(* CoDeSys 2.3.9.50 project: dacha.pro *)
(* Libraries: standard.lib 5.6.98 11:03:02, TcpIp.lib 9.1.14 13:33:22, TcBase.lib 14.5.09 11:14:08, TcSystem.lib 7.6.16 10:01:22, ModbusRTU.lib 13.5.15 12:38:16, TcIoFunctions.lib 27.1.17 16:22:22, COMlibV2.lb6 25.2.14 08:37:08, TcUtilities.lib 3.2.16 15:08:58 *)

(* Task configuration *)
TASK Standard (PRIORITY := 0, INTERVAL := T#50ms);
	MAIN
END_TASK

(* Global variable list: Global_Variables *)
VAR_GLOBAL


	Clear					: ClearComBuffer;
	MB						: ModbusRtuMaster_KL6x22B;
	TxBufferCom1			: ComBuffer;
	RxBufferCom1			: ComBuffer;
	SerialLineControlCom1		: SerialLineControl;
	ReceiveDataCom1		: ReceiveData;
	SendDataCom1			: SendData;
	Merc_address			: BYTE:=97;
	Sensor_CO2_high	 		: BYTE;	(*Старший байт датчика MH-Z19B*)
	Sensor_CO2_low 			: BYTE;	(*Младший байт датчика MH-Z19B*)
	iobroker					: iobroker_Struct;
	MB_vars					: stMB;
	Mercury					: stMercury;


	HW_temp_first_floor					AT %IW40:WORD;	(* Датчик температуры 1 этаж *)
	HW_temp_second_floor				AT %IW42:WORD;	(* Датчик температуры 2 этаж *)
	HW_temp_underfloor					AT %IW44:WORD;	(* Датчик температуры подпол 1 этаж *)
	HW_temp_sport						AT %IW46:WORD;	(* Датчик температуры спортзал *)

	HW_temp_sport_underfloor				AT %IW48:WORD;	(* Датчик температуры подпол спортзал *)
	HW_temp_sauna						AT %IW50:WORD;	(* Датчик температуры сауна*)
	HW_temp_street						AT %IW52:WORD;	(* Датчик температуры улица *)
	HW_temp_vent						AT %IW54:WORD;	(* Датчик температуры притока вентиляции *)

	HW_PIR_terrasa						AT %IX56.0:BOOL;		(*PIR датчик терраса *)
	HW_PIR_zapad						AT %IX56.1:BOOL;		(*PIR датчик запад *)
	HW_PIR_vostok						AT %IX56.2:BOOL;		(*PIR датчик восток *)
	HW_PIR_sport						AT %IX56.3:BOOL;		(*PIR датчик спортзал *)

	HW_GERKON_drovnik					AT %IX56.4:BOOL;		(*Геркон дровник *)
	HW_GERKON_door					AT %IX56.5:BOOL;		(*Геркон дверь *)
	HW_sensor_smoke_1floor				AT %IX56.6:BOOL;		(*Датчик дыма 1 этаж *)
	HW_sensor_smoke_2floor				AT %IX56.7:BOOL;		(*Датчик дыма 2 этаж *)

	HW_button_light_terrasa				AT %IX57.0:BOOL;		(* Кнопка прожектор терраса  *)
	HW_button_security					AT %IX57.1:BOOL;		(* Кнопка охрана  *)
	HW_button_vorota						AT %IX57.2:BOOL;		(* Кнопка открытия ворот  *)
	HW_button_kalitka					AT %IX57.3:BOOL;		(* Кнопка открытия калитки  *)

	HW_button_poliv_terrasa				AT %IX57.4:BOOL;		(* Кнопка полив терраса 2 часа  *)
	HW_button_poliv_zapad				AT %IX57.5:BOOL;		(* Кнопка полив запад  2 часа  *)
	HW_button_poliv_south				AT %IX57.6:BOOL;		(* Кнопка полив юг 2 часа  *)
(*	HW_reserved						AT %IX57.7:BOOL;	*)	(*   *)

	HW_sensor_supply					AT %IX58.0:BOOL;		(* Датчик напряжение  *)


	HW_heat_first_floor					AT %QX0.0:BOOL;		(* Отопление 1 этаж *)
	HW_heat_second_floor				AT %QX0.1:BOOL;		(* Отопление 2 этаж *)
	HW_heat_sport						AT %QX0.2:BOOL;		(* Отопление спортзал *)
	HW_heat_underfloor					AT %QX0.3:BOOL;		(* Отопление подпол *)
	HW_heat_sauna						AT %QX0.4:BOOL;		(* Отопление сауна *)
	HW_heat_bathroom					AT %QX0.5:BOOL;		(* Отопление душевая *)
	HW_heat_pipe						AT %QX0.6:BOOL;		(* Отопление водопровод *)
	HW_vent_underfloor					AT %QX0.7:BOOL;		(* Вентиляция подпола *)

	HW_vorota							AT %QX1.0:BOOL;		(* Ворота *)
	HW_kalitka							AT %QX1.1:BOOL;		(* Калитка *)
	HW_pomp_house						AT %QX1.2:BOOL;		(* Насос водоснабжения дома *)
	HW_pomp_garden					AT %QX1.3:BOOL;		(* Насос полива *)
	HW_light_garden						AT %QX1.4:BOOL;		(* Прожектор двор *)
	HW_light_terrasa						AT %QX1.5:BOOL;		(* Свет терраса *)
	HW_switch_security					AT %QX1.6:BOOL;		(* Реле охрана *)
	HW_switch_RS485					AT %QX1.7:BOOL:=TRUE;		(* RS485 line *)


	HW_vent_valve_input					AT %QX2.0:BOOL;		(* Клапан приточной вентиляции *)
	HW_vent_valve_output					AT %QX2.1:BOOL;		(* Клапан вытяжной вентиляции *)
	HW_trans_power						AT %QX2.2:BOOL;		(*Подача тока на трансформатор и реле ТЭН-а *)
	HW_vent_in_heat						AT %QX2.3:BOOL;		(* Подогрев притока - ТЭН *)
	HW_vent_in_heat_level				AT %QX2.4:BOOL;		(* Подогрев притока ночной режим   -5 К ТЭН *)
	HW_vent_in_trans_105_130				AT %QX2.5:BOOL:=FALSE;  (* Напряжение 110 или 130 В *)
	HW_vent_in_trans_160_220				AT %QX2.6:BOOL:=FALSE;  (* Напряжение 160 или 220 В *)
	HW_vent_in_trans_LO_HI				AT %QX2.7:BOOL:=FALSE;  (* Напряжение 110/130  или 160/220 В *)

	HW_poliv_terrasa						AT %QX3.0:BOOL;		(* полив терраса  *)
	HW_poliv_zapad						AT %QX3.1:BOOL;		(* полив запад   *)
	HW_poliv_south						AT %QX3.2:BOOL;		(* полив юг   *)


END_VAR

(* Global variable list: Global_Variables_persistent *)
VAR_GLOBAL PERSISTENT

	(*USER VARIABLES NEED TO BE ATTACHED TO %Q TO ENABLE SAVE IT IN NOVRAM, FOR CX ONLY *)

	Target_CO2_mem					AT %Q*:		INT;

	First_floor_temp_target_mem		AT %Q*:		INT;
	Second_floor_temp_target_mem		AT %Q*:		INT;
	Sport_temp_target_mem			AT %Q*:		INT;
	Sauna_temp_target_mem			AT %Q*:		INT;
	Underfloor_temp_target_mem		AT %Q*:		INT;
	Underfloor_humidity_target_mem	AT %Q*:		INT;

	Pomp_house_mem				AT %Q*:		BOOL;
	Pomp_garden_mem				AT %Q*:		BOOL;

	Light_garden_mem				AT %Q*:		BOOL;

	Vent_mem						AT %Q*:		BOOL;
	Vent_heat_mem					AT %Q*:		INT;
	Vent_heat_level_mem				AT %Q*:		BOOL;


END_VAR

(* Global variable list: TwinCAT_Configuration *)
(* Generated automatically by TwinCAT - (read only) *)
VAR_CONFIG
	.MB.InData AT %IB60 : MB_KL6inData22B;
	.MB.OutData AT %QB32 : MB_KL6outData22B;
	.Target_CO2_mem AT %QB6 : INT;
	.First_floor_temp_target_mem AT %QB56 : INT;
	.Second_floor_temp_target_mem AT %QB60 : INT;
	.Sport_temp_target_mem AT %QB62 : INT;
	.Sauna_temp_target_mem AT %QB72 : INT;
	.Underfloor_temp_target_mem AT %QB64 : INT;
	.Underfloor_humidity_target_mem AT %QB76 : INT;
	.Pomp_house_mem AT %QX68.0 : BOOL;
	.Pomp_garden_mem AT %QX74.0 : BOOL;
	.Light_garden_mem AT %QX66.1 : BOOL;
	.Vent_mem AT %QX28.0 : BOOL;
	.Vent_heat_mem AT %QB8 : INT;
	.Vent_heat_level_mem AT %QX28.3 : BOOL;
END_VAR

(* Global variable list: Variable_Configuration *)
VAR_CONFIG
	MB.InData AT %IB12 : MB_KL6inData22B;
	MB.OutData AT %QB12 : MB_KL6outData22B;

END_VAR

(* Data type *)
TYPE iobroker_Struct  :
STRUCT
	Vent_status				: 	INT;
	Valve_status				: 	INT;
	First_floor_temp 			:	REAL;
	First_floor_temp_target 		:	INT;
	First_floor_hum 			:	REAL;
	First_floor_CO2			:	REAL;
	Kitchen_room_temp		:	REAL;
	Kitchen_room_hum		:	REAL;
	Second_floor_temp 		:	REAL;
	Second_floor_temp_target 	:	INT;
	Second_floor_CO2 		:	REAL;
	Sport_temp	 			:	REAL;
	Sport_temp_target			:	INT;
	Sauna_temp	 			:	REAL;
	Sauna_temp_target		:	INT;
	Underfloor_temp			:	REAL;
	Underfloor_temp_target	:	INT;
	Underfloor_humidity		:	REAL;
	Underfloor_humidity_target	:	INT;
	Sport_underfloor_temp		:	REAL;
	Street_temp				:	REAL;
	Vent_temp				:	REAL;
	PIR_terrasa				:	BOOL:=TRUE;
	PIR_zapad				:	BOOL:=TRUE;
	PIR_vostok				:	BOOL:=TRUE;
	PIR_sport				:	BOOL:=TRUE;
	GERKON_drovnik			:	BOOL:=TRUE;
	Vent_input_level			:	INT;  (*  0-220 V  *)
	Vent_output_level			:	INT; (*0-100%*)
	Temp_vent_in			:	REAL;
	Vent_valve_status			:	INT;
	Security_status			:	BOOL;
	Target_CO2				:	INT;
	Vent						:	BOOL;
	Vent_underfloor			:	BOOL;
	Vent_out					:	BOOL;
	Vent_heat				:	INT;
	Vent_heat_level			:	BOOL;
	Vorota					:	BOOL;
	Vorota_open				:	BOOL;
	Kalitka					:	BOOL;
	Smoke					:	BOOL;
	Sensor_supply			:	BOOL;
	Pomp_house				:	BOOL;
	Pomp_garden			:	BOOL;
	Light_garden				:	BOOL;
	Poliv_zapad				:	BOOL;
	Poliv_terrasa				:	BOOL;
	Poliv_south				:	BOOL;
	Poliv_zapad_minutes		:	INT;
	Poliv_terrasa_minutes		:	INT;
	Poliv_south_minutes		:	INT;
	Uv1						:	REAL;
	Uv2						:	REAL;
	Uv3						:	REAL;
	Pw1						:	REAL;
	Pw2						:	REAL;
	Pw3						:	REAL;
	Pw_total					:	REAL;
	Ia1						:	REAL;
	Ia2						:	REAL;
	Ia3						:	REAL;
	E_T1					:	REAL;
	E_T2					:	REAL; (* 64 values*)

(*	M1T1					:	DWORD:=0;
	M1T2					:	DWORD:=0; (* 66 values*)

	M2T1					:	DWORD:=0; (* 67 values*)
	M2T2					:	DWORD:=0;
	M3T1					:	DWORD:=0;
	M3T2					:	DWORD:=0;
	M4T1					:	DWORD:=0; (* 70 values*)
	M4T2					:	DWORD:=0;
	M5T1					:	DWORD:=0;
	M5T2					:	DWORD:=0;
	M6T1					:	DWORD:=0;
	M6T2					:	DWORD:=0;
	M7T1					:	DWORD:=0;
	M7T2					:	DWORD:=0;
	M8T1					:	DWORD:=0;
	M8T2					:	DWORD:=0;
	M9T1					:	DWORD:=0;
	M9T2					:	DWORD:=0;
	M10T1					:	DWORD:=0;
	M10T2					:	DWORD:=0;
	M11T1					:	DWORD:=0;
	M11T2					:	DWORD:=0;
	M12T1					:	DWORD:=0;
	M12T2					:	DWORD:=0;   (* 86 values*)
*)

END_STRUCT
END_TYPE

(* Data type *)
(* @NESTEDCOMMENTS := 'Yes' *)
(* @PATH := '' *)
(* @OBJECTFLAGS := '0, 8' *)
TYPE ST_MqttReceivedPublishTelegram :
STRUCT
	sTopic		: STRING[255];
	sValue		: STRING[255];
	bHasData	: BOOL;
END_STRUCT
END_TYPE
(* @END_DECLARATION := '0' *)

(* Data type *)
(* @NESTEDCOMMENTS := 'Yes' *)
(* @PATH := '' *)
(* @OBJECTFLAGS := '0, 8' *)
TYPE ST_MqttSettings :
STRUCT
	(* informations *)
	sMqttClientId	: STRING[23];
	sMqttUserId	: STRING[25];
	sMqttPassword	: STRING[25];
	sMqttBrokerIP	: STRING[15];
	nMqttBrokerPort	: UDINT := 1883;

	(* state *)
	bSocketConnection	: BOOL := FALSE;
	bConnected			: BOOL := FALSE;
	bConnectPackageSent	: BOOL := FALSE;
	bDisconnect			: BOOL := FALSE;
	bError				: BOOL := FALSE;
	bValidConnection	: BOOL := FALSE;
	bActive				: BOOL := FALSE;
	wPackageIdentifier	: WORD := 1;
	hSocket				: T_HSOCKET;
	tonSendPingReq		: TON;

	(* send *)
	stMqttSendTelegram			: ST_MqttTelegram;
	stMqttLastSendTelegram		: ST_MqttTelegram;

	(* receive *)
	stMqttReceivedTelegram			: ST_MqttTelegram;
	stMqttLastReceivedTelegram		: ST_MqttTelegram;
	stMqttReceivedPublishTelegram	: ST_MqttReceivedPublishTelegram;

	(* settings internal *)
	iTelegramSize	: INT := 544;
	usKeepAliveTime	: USINT := 60; (* seconds *)

END_STRUCT
END_TYPE
(* @END_DECLARATION := '0' *)

(* Data type *)
(* @NESTEDCOMMENTS := 'Yes' *)
(* @PATH := '' *)
(* @OBJECTFLAGS := '0, 8' *)
TYPE ST_MqttTelegram :
STRUCT
	arMqttData 	: ARRAY[0..544] OF BYTE;
	nDataLength	: UDINT := 0;
END_STRUCT
END_TYPE
(* @END_DECLARATION := '0' *

(* Data type *)
TYPE stMB :
STRUCT

	M1T1							AT %MW0	:REAL;  (* modbus address 12288 *)
	M1T2							AT %MW4	:REAL;
	M2T1							AT %MW8	:REAL;
	M2T2							AT %MW12	:REAL;
	M3T1							AT %MW16	:REAL;
	M3T2							AT %MW20	:REAL;
	M4T1							AT %MW24	:REAL;
	M4T2							AT %MW28	:REAL;
	M5T1							AT %MW32	:REAL;
	M5T2							AT %MW36	:REAL;
	M6T1							AT %MW40	:REAL;
	M6T2							AT %MW44	:REAL;
	M7T1							AT %MW48	:REAL;
	M7T2							AT %MW52	:REAL;
	M8T1							AT %MW56	:REAL;
	M8T2							AT %MW60	:REAL;
	M9T1							AT %MW64	:REAL;
	M9T2							AT %MW68	:REAL;
	M10T1							AT %MW72	:REAL;
	M10T2							AT %MW76	:REAL;
	M11T1							AT %MW80	:REAL;
	M11T2							AT %MW84	:REAL;
	M12T1							AT %MW88	:REAL;
	M12T2							AT %MW92	:REAL;

END_STRUCT
END_TYPE

(* Data type *)
TYPE stMercury :
STRUCT

	M1T1					:	REAL;
	M1T2					:	REAL;
	M2T1					:	REAL;
	M2T2					:	REAL;
	M3T1					:	REAL;
	M3T2					:	REAL;
	M4T1					:	REAL;
	M4T2					:	REAL;
	M5T1					:	REAL;
	M5T2					:	REAL;
	M6T1					:	REAL;
	M6T2					:	REAL;
	M7T1					:	REAL;
	M7T2					:	REAL;
	M8T1					:	REAL;
	M8T2					:	REAL;
	M9T1					:	REAL;
	M9T2					:	REAL;
	M10T1					:	REAL;
	M10T2					:	REAL;
	M11T1					:	REAL;
	M11T2					:	REAL;
	M12T1					:	REAL;
	M12T2					:	REAL;

END_STRUCT
END_TYPE

(* POU MAIN, ST *)
PROGRAM MAIN
VAR

	INITVAR					: BOOL:=FALSE;

END_VAR
IF (INITVAR=FALSE) THEN

	(* START RESTORE VARS FROM MEMORY AFTER REBOOT/RESET/LOST POWER *)

	iobroker.Target_CO2				:=	Target_CO2_mem;
	iobroker.First_floor_temp_target		:=	First_floor_temp_target_mem;
	iobroker.Second_floor_temp_target	:=	Second_floor_temp_target_mem;
	iobroker.Sport_temp_target			:=	Sport_temp_target_mem;
	iobroker.Sauna_temp_target		:=	Sauna_temp_target_mem;

	iobroker.Underfloor_temp_target		:=	Underfloor_temp_target_mem;
	iobroker.Underfloor_humidity_target	:=	Underfloor_humidity_target_mem;
	iobroker.Vent						:=	Vent_mem;
	iobroker.Vent_heat				:=	Vent_heat_mem;
	iobroker.Vent_heat_level			:=	Vent_heat_level_mem;
	iobroker.Pomp_house				:=	Pomp_house_mem;
	iobroker.Pomp_garden				:=	Pomp_garden_mem;
	iobroker.Light_garden				:=	Light_garden_mem;
	(* END RESTORE VARS FROM MEMORY AFTER REBOOT/RESET/LOST POWER *)

	INITVAR:=TRUE;
ELSE
	(*START SAVE VARS to PERSISTENT MEMORY*)
	Target_CO2_mem					:=	iobroker.Target_CO2;
	First_floor_temp_target_mem		:=	iobroker.First_floor_temp_target;
	Second_floor_temp_target_mem		:=	iobroker.Second_floor_temp_target;
	Sport_temp_target_mem			:=	iobroker.Sport_temp_target;
	Underfloor_temp_target_mem		:=	iobroker.Underfloor_temp_target;
	Underfloor_humidity_target_mem	:=	iobroker.Underfloor_humidity_target;
	Vent_mem						:=	iobroker.Vent;
	Vent_heat_mem					:=	iobroker.Vent_heat;
	Vent_heat_level_mem				:=	iobroker.Vent_heat_level;
	Light_garden_mem				:=	iobroker.Light_garden;
	Pomp_house_mem				:=	iobroker.Pomp_house;
	(*END SAVE VARS to PERSISTENT MEMORY*)


	Sensors;						(* Аналогвые датчики на шине KL *)
	Security;						(* Мониторинг датчиков охраны *)
	RS485read;					(* Опрос устройств на шине RS485 *)
	Mqtt;						(* MQTT *)
	Thermocontrol;				(* Термостат*)
	VentControl;					(* Глобальный контроль вентустановки*)
	VentPower;					(* Авторегулировка мощности вентустановки по датчикам CO2*)
	Poliv;						(* Таймеры зонального полива *)


	(* Прямое присовение виртуальных переменных к переменным, жестко привязаным к физ. портам. Частота обновления= циклу ПЛК (50 мсек) : *)
	HW_vorota					:=	iobroker.Vorota;
	HW_kalitka					:=	iobroker.Kalitka;
	HW_pomp_house				:=	iobroker.Pomp_house;
	HW_light_garden				:=	iobroker.Light_garden;
	iobroker.Sensor_supply		:=	HW_sensor_supply;
	HW_vent_underfloor			:=	iobroker.Vent_underfloor;

END_IF
END_PROGRAM

(* POU Sensors, ST *)
PROGRAM Sensors
VAR
	Period_sensors_read		: INT:=30; (* Частота присвоения значений аналоговых температурных датчиков с модулей KL, секунды *)
	Timer					: TON;
	TimerQ					: BOOL;
	tTimerValue				: TIME;
END_VAR
Timer();

tTimerValue := DINT_TO_TIME(Period_sensors_read*1000);

	Timer(IN:=NOT TimerQ , PT:=tTimerValue , Q=>TimerQ , ET=> );
	IF timer.q THEN

		(*Temperature First_floor start*)
		iobroker.First_floor_temp:=WORD_TO_REAL(HW_temp_first_floor);
		IF (iobroker.First_floor_temp/10>1000)  THEN
			iobroker.First_floor_temp:=iobroker.First_floor_temp-65535;
			iobroker.First_floor_temp:=iobroker.First_floor_temp/10;
		ELSE
			iobroker.First_floor_temp:=iobroker.First_floor_temp/10;
		END_IF
		(*Temperature First_floor end*)

		(*Temperature second_floor start*)
		iobroker.Second_floor_temp:=WORD_TO_REAL(HW_temp_second_floor);
		IF (iobroker.Second_floor_temp/10>1000)  THEN
			iobroker.Second_floor_temp:=iobroker.Second_floor_temp-65535;
			iobroker.Second_floor_temp:=iobroker.Second_floor_temp/10;
		ELSE
			iobroker.Second_floor_temp:=iobroker.Second_floor_temp/10;
		END_IF
		(*Temperature second_floor end*)

		(*Temperature second_floor start*)
		iobroker.Sport_temp:=WORD_TO_REAL(HW_temp_sport);
		IF (iobroker.Sport_temp/10>1000)  THEN
			iobroker.Sport_temp:=iobroker.Sport_temp-65535;
			iobroker.Sport_temp:=iobroker.Sport_temp/10;
		ELSE
			iobroker.Sport_temp:=iobroker.Sport_temp/10;
		END_IF
		(*Temperature second_floor end*)

		(*Temperature street start*)
		iobroker.Street_temp:=WORD_TO_REAL(HW_temp_street);
		IF (iobroker.Street_temp/10>1000)  THEN
			iobroker.Street_temp:=iobroker.Street_temp-65535;
			iobroker.Street_temp:=iobroker.Street_temp/10;
		ELSE
			iobroker.Street_temp:=iobroker.Street_temp/10;
		END_IF
		(*Temperature street end*)

		(*Temperature vent start*)
		iobroker.Vent_temp:=WORD_TO_REAL(HW_temp_vent);
		IF (iobroker.Vent_temp/10>1000)  THEN
			iobroker.Vent_temp:=iobroker.Vent_temp-65535;
			iobroker.Vent_temp:=iobroker.Vent_temp/10;
		ELSE
			iobroker.Vent_temp:=iobroker.Vent_temp/10;
		END_IF
		(*Temperature vent end*)
	END_IF
END_PROGRAM

(* POU Security, ST *)
PROGRAM Security
VAR
	TRIG_PIR_terrasa			:	F_TRIG;
	TRIG_PIR_zapad			:	F_TRIG;
	TRIG_PIR_vostok			:	F_TRIG;
	TRIG_PIR_sport			:	F_TRIG;
	TRIG_GERKON_drovnik	:	F_TRIG;
	TRIG_sensor_smoke_1floor:	F_TRIG;

	trig_mem_terrasa				:	BOOL:=FALSE;
	trig_mem_zapad				:	BOOL:=FALSE;
	trig_mem_vostok				:	BOOL:=FALSE;
	trig_mem_sport				:	BOOL:=FALSE;
	trig_mem_drovnik				:	BOOL:=FALSE;
	trig_mem_sensor_smoke_1floor	:	BOOL:=FALSE;

END_VAR
(*  Используем триггеры для исключения ложной информации о сработке датчиков при перезагрузке ПЛК *)


TRIG_PIR_terrasa(CLK :=HW_PIR_terrasa);
TRIG_PIR_zapad(CLK :=HW_PIR_zapad);
TRIG_PIR_vostok(CLK :=HW_PIR_vostok);
TRIG_PIR_sport(CLK :=HW_PIR_sport);
TRIG_GERKON_drovnik(CLK :=HW_GERKON_drovnik);
TRIG_sensor_smoke_1floor(CLK :=HW_sensor_smoke_1floor);


IF (NOT TRIG_PIR_terrasa.Q) THEN
	iobroker.PIR_terrasa:=NOT TRIG_PIR_terrasa.Q;
END_IF
IF (trig_mem_terrasa=TRUE) THEN
	iobroker.PIR_terrasa:=FALSE;
	trig_mem_terrasa:=FALSE;
END_IF
IF (TRIG_PIR_terrasa.Q) THEN
	trig_mem_terrasa:=TRUE;
END_IF



IF (NOT TRIG_PIR_zapad.Q) THEN
	iobroker.PIR_zapad:=NOT TRIG_PIR_zapad.Q;
END_IF
IF (trig_mem_zapad=TRUE) THEN
	iobroker.PIR_zapad:=FALSE;
	trig_mem_zapad:=FALSE;
END_IF
IF (TRIG_PIR_zapad.Q) THEN
	trig_mem_zapad:=TRUE;
END_IF


IF (NOT TRIG_PIR_vostok.Q) THEN
	iobroker.PIR_vostok:=NOT TRIG_PIR_vostok.Q;
END_IF
IF (trig_mem_vostok=TRUE) THEN
	iobroker.PIR_vostok:=FALSE;
	trig_mem_vostok:=FALSE;
END_IF
IF (TRIG_PIR_vostok.Q) THEN
	trig_mem_vostok:=TRUE;
END_IF


IF (NOT TRIG_PIR_sport.Q) THEN
	iobroker.PIR_sport:=NOT TRIG_PIR_sport.Q;
END_IF
IF (trig_mem_sport=TRUE) THEN
	iobroker.PIR_sport:=FALSE;
	trig_mem_sport:=FALSE;
END_IF
IF (TRIG_PIR_sport.Q) THEN
	trig_mem_sport:=TRUE;
END_IF

IF (NOT TRIG_GERKON_drovnik.Q) THEN
	iobroker.GERKON_drovnik:=NOT TRIG_GERKON_drovnik.Q;
END_IF
IF (trig_mem_drovnik=TRUE) THEN
	iobroker.GERKON_drovnik:=FALSE;
	trig_mem_drovnik:=FALSE;
END_IF
IF (TRIG_GERKON_drovnik.Q) THEN
	trig_mem_drovnik:=TRUE;
END_IF


IF (NOT TRIG_sensor_smoke_1floor.Q) THEN
	iobroker.SMOKE:=NOT TRIG_sensor_smoke_1floor.Q;
END_IF
IF (trig_mem_sensor_smoke_1floor=TRUE) THEN
	iobroker.SMOKE:=FALSE;
	trig_mem_sensor_smoke_1floor:=FALSE;
END_IF
IF (TRIG_sensor_smoke_1floor.Q) THEN
	trig_mem_sensor_smoke_1floor:=TRUE;
END_IF
END_PROGRAM

(* POU RS485read, ST *)
PROGRAM RS485read
VAR

	password_1				: ARRAY [1..6] OF BYTE:=6(1); (* пароль к меркуриям, по умолчанию 6 единиц*)
	crctest					: WORD;
	arrReceive				: ARRAY[1..22] OF BYTE;
	arrSend					: ARRAY[1..22] OF BYTE;

	MBdata_kitchen			 : ARRAY [1..2] OF WORD;
	FtrigBusy				: F_TRIG;
	timeoutvalue				: TIME := T#500ms;		(* timeout while waiting for an answer of the modbus slave *)
	state					: INT;
	busy					: BOOL;
	LastErrorstate				: INT;
	LastModbusError			: ST_ModbusErrorDiagnostics;
	CounterError				: DINT;
	CounterSuccess			: DINT;
	Timer1					: TON;
	Timer1Q					: BOOL;
	Timer_day				:TON;
	Timer_dayQ				:BOOL;

	tmCheck					:TON;

	get_co2_mh_z19b_1floor	: FB_GET_CO2_MH_Z19B;
	get_co2_mh_z19b_2floor	: FB_GET_CO2_MH_Z19B;
	get_supply				: FB_GET_SUPPLY;
	get_current				: FB_GET_CURRENT;
	get_power				: FB_GET_POWER;
	get_energy_E_T1			: FB_GET_ENERGY;
	get_energy_E_T2			: FB_GET_ENERGY;
	get_energy_M1T1			: FB_GET_ENERGY;
	get_energy_M1T2			: FB_GET_ENERGY;
	get_energy_M2T1			: FB_GET_ENERGY;
	get_energy_M2T2			: FB_GET_ENERGY;
	get_energy_M3T1			: FB_GET_ENERGY;
	get_energy_M3T2			: FB_GET_ENERGY;
	get_energy_M4T1			: FB_GET_ENERGY;
	get_energy_M4T2			: FB_GET_ENERGY;
	get_energy_M5T1			: FB_GET_ENERGY;
	get_energy_M5T2			: FB_GET_ENERGY;
	get_energy_M6T1			: FB_GET_ENERGY;
	get_energy_M6T2			: FB_GET_ENERGY;
	get_energy_M7T1			: FB_GET_ENERGY;
	get_energy_M7T2			: FB_GET_ENERGY;
	get_energy_M8T1			: FB_GET_ENERGY;
	get_energy_M8T2			: FB_GET_ENERGY;
	get_energy_M9T1			: FB_GET_ENERGY;
	get_energy_M9T2			: FB_GET_ENERGY;
	get_energy_M10T1		: FB_GET_ENERGY;
	get_energy_M10T2		: FB_GET_ENERGY;
	get_energy_M11T1		: FB_GET_ENERGY;
	get_energy_M11T2		: FB_GET_ENERGY;
	get_energy_M12T1		: FB_GET_ENERGY;
	get_energy_M12T2		: FB_GET_ENERGY;

	get_co2_mh_z19b_1floor_done	: BOOL;
	get_co2_mh_z19b_2floor_done	: BOOL;
	get_supply_done			: BOOL;
	get_current_done			: BOOL;
	get_power_done			: BOOL;
	get_energy_E_T1_done	: BOOL;
	get_energy_E_T2_done	: BOOL;
	get_energy_M1T1_done	: BOOL;
	get_energy_M1T2_done	: BOOL;
	get_energy_M2T1_done	: BOOL;
	get_energy_M2T2_done	: BOOL;
	get_energy_M3T1_done	: BOOL;
	get_energy_M3T2_done	: BOOL;
	get_energy_M4T1_done	: BOOL;
	get_energy_M4T2_done	: BOOL;
	get_energy_M5T1_done	: BOOL;
	get_energy_M5T2_done	: BOOL;
	get_energy_M6T1_done	: BOOL;
	get_energy_M6T2_done	: BOOL;
	get_energy_M7T1_done	: BOOL;
	get_energy_M7T2_done	: BOOL;
	get_energy_M8T1_done	: BOOL;
	get_energy_M8T2_done	: BOOL;
	get_energy_M9T1_done	: BOOL;
	get_energy_M9T2_done	: BOOL;
	get_energy_M10T1_done	: BOOL;
	get_energy_M10T2_done	: BOOL;
	get_energy_M11T1_done	: BOOL;
	get_energy_M11T2_done	: BOOL;
	get_energy_M12T1_done	: BOOL;
	get_energy_M12T2_done	: BOOL;
END_VAR

VAR_INPUT


END_VAR
tmCheck();
Timer_day();

CASE state OF
	0:
		MB.ReadRegs(Execute:= FALSE);

		state := 1;
	1:	(* Read Temp and Hum data  from sensor *)
		Clear(Buffer := RxBufferCom1);
		MB.ReadRegs(
			UnitID:= 16#07, (* station address *)
			Quantity:= 2,	(* WORDs *)
			MBAddr:= 0,
			cbLength:= 6,
			pMemoryAddr:= ADR(MBdata_kitchen),
			Execute:= TRUE,
			Timeout:= timeoutvalue,
			Busy => busy,
		);
		IF NOT busy THEN
			IF (mb.Error = FALSE ) THEN
				iobroker.Kitchen_room_temp:=WORD_TO_REAL(MBdata_kitchen[1])/10;
				iobroker.Kitchen_room_hum:=WORD_TO_REAL(MBdata_kitchen[2])/10;
				MB.ReadRegs(Execute:= FALSE);
				state := 2;
			END_IF
			MB.ReadRegs(Execute:= FALSE);
			state :=2;
		END_IF

2:	(* Read CO2 from sensor *)

		tmCheck(in:=FALSE);
		tmCheck(in:=TRUE,pt:=t#2s);
		get_co2_mh_z19b_1floor_done := FALSE;
		get_co2_mh_z19b_1floor( co2=>iobroker.First_Floor_CO2, done=>get_co2_mh_z19b_1floor_done);
		IF get_co2_mh_z19b_1floor_done = TRUE THEN
			state:=3;
		ELSIF tmcheck.Q THEN
			 state:=3;
		END_IF

3:
	HW_switch_RS485:=TRUE;
	Timer1(IN:=NOT Timer1Q , PT:=T#1s , Q=>Timer1Q , ET=> );
	IF timer1.q THEN
		state:=4;
	END_IF

4:

		tmCheck(in:=FALSE);
		tmCheck(in:=TRUE,pt:=t#2s);
		get_co2_mh_z19b_2floor_done := FALSE;
		get_co2_mh_z19b_2floor( co2=>iobroker.Second_Floor_CO2, done=>get_co2_mh_z19b_2floor_done);
		IF get_co2_mh_z19b_2floor_done = TRUE THEN
			state:=41;
		ELSIF tmcheck.Q THEN
			 state:=41;
		END_IF



41:
	Timer1(IN:=NOT Timer1Q , PT:=T#2s , Q=>Timer1Q , ET=> );
	IF timer1.q THEN
	HW_switch_RS485:=FALSE;
		state:=5;
	END_IF

5: (*открываем канал*)


	Clear(Buffer := RxBufferCom1);
	arrSend[1]:=Merc_address;
	arrSend[2]:=1; (*код доступа*)
	arrSend[3]:=1; (*Уровень доступа*)

	MEMCPY(ADR(arrSend)+3,ADR(password_1),6); (*пароль*)
	crctest:=F_CRC16(ADR(arrSend),9); (*расчет контрольной суммы*)
	MEMCPY(ADR(arrSend)+9,ADR(crctest),SIZEOF(crctest)); (*прибавление контрольной суммы к запросу*)
	SendDataCom1(pSendData:=ADR(arrSend),Length:=11,TXBuffer:=TxBufferCom1,Busy=>,Error=>);
	tmCheck(in:=FALSE); tmCheck(in:=TRUE,pt:=t#2s); 	(*запуск таймера проверки - потеря связи\обрыв кабеля*)
	state:=6;

6: (*ответ*)
	ReceiveDataCom1(pPrefix:=,LenPrefix:=,pSuffix:=,LenSuffix:=,
	pReceiveData:=ADR(arrReceive),SizeReceiveData:=4,
	Timeout:=t#2s,Reset:=,
	RXbuffer:=RxBufferCom1,
	DataReceived=>,busy=>,Error=>,RxTimeout=>,LenReceiveData=>);
	IF ReceiveDataCom1.Error <> 0 THEN state:=888; END_IF
	IF receiveDataCom1.DataReceived THEN state:=7;
	ELSIF tmcheck.Q THEN state:=888;
	END_IF
7: (*проверка ответа*)

	IF arrReceive[1] = Merc_address THEN state:= 8;
	ELSE	state:=888;
	END_IF



8:
		tmCheck(in:=FALSE);
		tmCheck(in:=TRUE,pt:=t#2s);
		get_supply_done := FALSE;
		get_supply( byte1:=16#8, byte2:=16#16, byte3:=16#11,  supply1=>iobroker.UV1,supply2=>iobroker.UV2,supply3=>iobroker.UV3, done=>get_supply_done);
		IF get_supply_done = TRUE THEN
			state:=9;
		ELSIF tmcheck.Q THEN
			 state:=888;
		END_IF

 (*запрос на чтение тока  на всех фазах
--------------------------------------------------------------------------------------------------------------------------------------------------------------------
*)
9:
		tmCheck(in:=FALSE);
		tmCheck(in:=TRUE,pt:=t#2s);
		get_current_done := FALSE;
		get_current(byte1:=16#8, byte2:=16#16, byte3:=16#21,  current1=>iobroker.Ia1,current2=>iobroker.Ia2,current3=>iobroker.Ia3, done=>get_current_done);
		IF get_current_done = TRUE THEN
			state:=10;
		ELSIF tmcheck.Q THEN state:=888;
		END_IF

 (*запрос на чтение мощности  на всех фазах
--------------------------------------------------------------------------------------------------------------------------------------------------------------------
*)

10:
		tmCheck(in:=FALSE);
		tmCheck(in:=TRUE,pt:=t#2s);
		get_power_done := FALSE;
		get_power(byte1:=16#8, byte2:=16#16, byte3:=16#0,  power_total=>iobroker.pw_total, power1=>iobroker.pw1, power2=>iobroker.pw2,power3=>iobroker.pw3,done=>get_power_done);
		IF get_power_done = TRUE THEN
			state:=11;
		ELSIF tmcheck.Q THEN state:=888;
		END_IF

 (*запрос на чтение энергии T1
--------------------------------------------------------------------------------------------------------------------------------------------------------------------
*)
11:
	tmCheck(in:=FALSE);
		tmCheck(in:=TRUE,pt:=t#2s);
		get_energy_E_T1_done := FALSE;
		get_energy_E_T1(byte1:=5, byte2:=16#0, byte3:=1,  energy=>iobroker.E_T1, done=>get_energy_E_T1_done);
		IF get_energy_E_T1_done = TRUE THEN
			state:=12;
		ELSIF tmcheck.Q THEN state:=888;
		END_IF
 (*запрос на чтение энергии T2
--------------------------------------------------------------------------------------------------------------------------------------------------------------------
*)

12:
	tmCheck(in:=FALSE);
		tmCheck(in:=TRUE,pt:=t#2s);
		get_energy_E_T2_done := FALSE;
		get_energy_E_T2(byte1:=5, byte2:=16#0, byte3:=2,  energy=>iobroker.E_T2, done=>get_energy_E_T2_done);
		IF get_energy_E_T2_done = TRUE THEN
			state:=13;
		ELSIF tmcheck.Q THEN state:=888;
		END_IF


13:
		Timer_day(IN:=NOT Timer_dayQ , PT:=T#10m , Q=>Timer_dayQ , ET=> );
			IF timer_day.q THEN
				state:=14;
			ELSE
				state:=888;
			END_IF

14:
		tmCheck(in:=FALSE);
		tmCheck(in:=TRUE,pt:=t#2s);
		get_energy_M1T1_done := FALSE;
		get_energy_M1T1(byte1:=5, byte2:=16#31, byte3:=1,   energy=>MB_vars.M1T1,done=>get_energy_M1T1_done);
		IF get_energy_M1T1_done = TRUE THEN
			Mercury.M1T1:=MB_vars.M1T1;
			state:=15;
		ELSIF tmcheck.Q THEN state:=888;
		END_IF
15:
		tmCheck(in:=FALSE);
		tmCheck(in:=TRUE,pt:=t#2s);
		get_energy_M1T2_done := FALSE;
		get_energy_M1T2(byte1:=5, byte2:=16#31, byte3:=2,energy=>MB_vars.M1T2,done=>get_energy_M1T2_done);
		IF get_energy_M1T2_done = TRUE THEN
			Mercury.M1T2:=MB_vars.M1T2;
			state:=16;
		ELSIF tmcheck.Q THEN state:=888;
		END_IF

16:
		tmCheck(in:=FALSE);
		tmCheck(in:=TRUE,pt:=t#2s);
		get_energy_M2T1_done := FALSE;
		get_energy_M2T1(byte1:=5, byte2:=16#32, byte3:=1, energy=>MB_vars.M2T1, done=>get_energy_M2T1_done);
		IF get_energy_M2T1_done = TRUE THEN
			Mercury.M2T1:=MB_vars.M2T1;
			state:=17;
		ELSIF tmcheck.Q THEN state:=888;
		END_IF
17:
		tmCheck(in:=FALSE);
		tmCheck(in:=TRUE,pt:=t#2s);
		get_energy_M2T2_done := FALSE;
		get_energy_M2T2(byte1:=5, byte2:=16#32, byte3:=2, energy=>MB_vars.M2T2,done=>get_energy_M2T2_done);
		IF get_energy_M2T2_done = TRUE THEN
			Mercury.M2T2:=MB_vars.M2T2;
			state:=18;
		ELSIF tmcheck.Q THEN state:=888;
		END_IF
18:
		tmCheck(in:=FALSE);
		tmCheck(in:=TRUE,pt:=t#2s);
		get_energy_M3T1_done := FALSE;
		get_energy_M3T1(byte1:=5, byte2:=16#33, byte3:=1, energy=>MB_vars.M3T1, done=>get_energy_M3T1_done);
		IF get_energy_M3T1_done = TRUE THEN
			Mercury.M3T1:=MB_vars.M3T1;
			state:=19;
		ELSIF tmcheck.Q THEN state:=888;
		END_IF
19:
		tmCheck(in:=FALSE);
		tmCheck(in:=TRUE,pt:=t#2s);
		get_energy_M3T2_done := FALSE;
		get_energy_M3T2(byte1:=5, byte2:=16#33, byte3:=2, energy=>MB_vars.M3T2,done=>get_energy_M3T2_done);
		IF get_energy_M3T2_done = TRUE THEN
			Mercury.M3T2:=MB_vars.M3T2;
			state:=20;
		ELSIF tmcheck.Q THEN state:=888;
		END_IF
20:
		tmCheck(in:=FALSE);
		tmCheck(in:=TRUE,pt:=t#2s);
		get_energy_M4T1_done := FALSE;
		get_energy_M4T1(byte1:=5, byte2:=16#34, byte3:=1, energy=>MB_vars.M4T1, done=>get_energy_M4T1_done);
		IF get_energy_M4T1_done = TRUE THEN
			Mercury.M4T1:=MB_vars.M4T1;
			state:=21;
		ELSIF tmcheck.Q THEN state:=888;
		END_IF
21:
		tmCheck(in:=FALSE);
		tmCheck(in:=TRUE,pt:=t#2s);
		get_energy_M4T2_done := FALSE;
		get_energy_M4T2(byte1:=5, byte2:=16#34, byte3:=2, energy=>MB_vars.M4T2,done=>get_energy_M4T2_done);
		IF get_energy_M4T2_done = TRUE THEN
			Mercury.M4T2:=MB_vars.M4T2;
			state:=22;
		ELSIF tmcheck.Q THEN state:=888;
		END_IF
22:
		tmCheck(in:=FALSE);
		tmCheck(in:=TRUE,pt:=t#2s);
		get_energy_M5T1_done := FALSE;
		get_energy_M5T1(byte1:=5, byte2:=16#35, byte3:=1, energy=>MB_vars.M5T1, done=>get_energy_M5T1_done);
		IF get_energy_M5T1_done = TRUE THEN
			Mercury.M5T1:=MB_vars.M5T1;
			state:=23;
		ELSIF tmcheck.Q THEN state:=888;
		END_IF
23:
		tmCheck(in:=FALSE);
		tmCheck(in:=TRUE,pt:=t#2s);
		get_energy_M5T2_done := FALSE;
		get_energy_M5T2(byte1:=5, byte2:=16#35, byte3:=2, energy=>MB_vars.M5T2,done=>get_energy_M5T2_done);
		IF get_energy_M5T2_done = TRUE THEN
			Mercury.M5T2:=MB_vars.M5T2;
			state:=24;
		ELSIF tmcheck.Q THEN state:=888;
		END_IF
24:
		tmCheck(in:=FALSE);
		tmCheck(in:=TRUE,pt:=t#2s);
		get_energy_M6T1_done := FALSE;
		get_energy_M6T1(byte1:=5, byte2:=16#36, byte3:=1, energy=>MB_vars.M6T1, done=>get_energy_M6T1_done);
		IF get_energy_M6T1_done = TRUE THEN
			Mercury.M6T1:=MB_vars.M6T1;
			state:=25;
		ELSIF tmcheck.Q THEN state:=888;
		END_IF
25:
		tmCheck(in:=FALSE);
		tmCheck(in:=TRUE,pt:=t#2s);
		get_energy_M6T2_done := FALSE;
		get_energy_M6T2(byte1:=5, byte2:=16#36, byte3:=2, energy=>MB_vars.M6T2,done=>get_energy_M6T2_done);
		IF get_energy_M6T2_done = TRUE THEN
			Mercury.M6T2:=MB_vars.M6T2;
			state:=26;
		ELSIF tmcheck.Q THEN state:=888;
		END_IF
26:
		tmCheck(in:=FALSE);
		tmCheck(in:=TRUE,pt:=t#2s);
		get_energy_M7T1_done := FALSE;
		get_energy_M7T1(byte1:=5, byte2:=16#37, byte3:=1, energy=>MB_vars.M7T1, done=>get_energy_M7T1_done);
		IF get_energy_M7T1_done = TRUE THEN
			Mercury.M7T1:=MB_vars.M7T1;
			state:=27;
		ELSIF tmcheck.Q THEN state:=888;
		END_IF
27:
		tmCheck(in:=FALSE);
		tmCheck(in:=TRUE,pt:=t#2s);
		get_energy_M7T2_done := FALSE;
		get_energy_M7T2(byte1:=5, byte2:=16#37, byte3:=2, energy=>MB_vars.M7T2,done=>get_energy_M7T2_done);
		IF get_energy_M7T2_done = TRUE THEN
			Mercury.M7T2:=MB_vars.M7T2;
			state:=28;
		ELSIF tmcheck.Q THEN state:=888;
		END_IF
28:
		tmCheck(in:=FALSE);
		tmCheck(in:=TRUE,pt:=t#2s);
		get_energy_M8T1_done := FALSE;
		get_energy_M8T1(byte1:=5, byte2:=16#38, byte3:=1, energy=>MB_vars.M8T1, done=>get_energy_M8T1_done);
		IF get_energy_M8T1_done = TRUE THEN
			Mercury.M8T1:=MB_vars.M8T1;
			state:=29;
		ELSIF tmcheck.Q THEN state:=888;
		END_IF
29:
		tmCheck(in:=FALSE);
		tmCheck(in:=TRUE,pt:=t#2s);
		get_energy_M8T2_done := FALSE;
		get_energy_M8T2(byte1:=5, byte2:=16#38, byte3:=2, energy=>MB_vars.M8T2,done=>get_energy_M8T2_done);
		IF get_energy_M8T2_done = TRUE THEN
			Mercury.M8T2:=MB_vars.M8T2;
			state:=30;
		ELSIF tmcheck.Q THEN state:=888;
		END_IF
30:
		tmCheck(in:=FALSE);
		tmCheck(in:=TRUE,pt:=t#2s);
		get_energy_M9T1_done := FALSE;
		get_energy_M9T1(byte1:=5, byte2:=16#39, byte3:=1, energy=>MB_vars.M9T1, done=>get_energy_M9T1_done);
		IF get_energy_M9T1_done = TRUE THEN
			Mercury.M9T1:=MB_vars.M9T1;
			state:=31;
		ELSIF tmcheck.Q THEN state:=888;
		END_IF
31:
		tmCheck(in:=FALSE);
		tmCheck(in:=TRUE,pt:=t#2s);
		get_energy_M9T2_done := FALSE;
		get_energy_M9T2(byte1:=5, byte2:=16#39, byte3:=2,  energy=>MB_vars.M9T2,done=>get_energy_M9T2_done);
		IF get_energy_M9T2_done = TRUE THEN
			Mercury.M9T2:=MB_vars.M9T2;
			state:=32;
		ELSIF tmcheck.Q THEN state:=888;
		END_IF
32:
		tmCheck(in:=FALSE);
		tmCheck(in:=TRUE,pt:=t#2s);
		get_energy_M10T1_done := FALSE;
		get_energy_M10T1(byte1:=5, byte2:=16#3A, byte3:=1,  energy=>MB_vars.M10T1, done=>get_energy_M10T1_done);
		IF get_energy_M10T1_done = TRUE THEN
			Mercury.M10T1:=MB_vars.M10T1;
			state:=33;
		ELSIF tmcheck.Q THEN state:=888;
		END_IF
33:
		tmCheck(in:=FALSE);
		tmCheck(in:=TRUE,pt:=t#2s);
		get_energy_M10T2_done := FALSE;
		get_energy_M10T2(byte1:=5, byte2:=16#3A, byte3:=2, energy=>MB_vars.M10T2,done=>get_energy_M10T2_done);
		IF get_energy_M10T2_done = TRUE THEN
			Mercury.M10T2:=MB_vars.M10T2;
			state:=34;
		ELSIF tmcheck.Q THEN state:=888;
		END_IF
34:
		tmCheck(in:=FALSE);
		tmCheck(in:=TRUE,pt:=t#2s);
		get_energy_M11T1_done := FALSE;
		get_energy_M11T1(byte1:=5, byte2:=16#3B, byte3:=1,  energy=>MB_vars.M11T1, done=>get_energy_M11T1_done);
		IF get_energy_M11T1_done = TRUE THEN
			Mercury.M11T1:=MB_vars.M11T1;
			state:=35;
		ELSIF tmcheck.Q THEN state:=888;
		END_IF
35:
		tmCheck(in:=FALSE);
		tmCheck(in:=TRUE,pt:=t#2s);
		get_energy_M11T2_done := FALSE;
		get_energy_M11T2(byte1:=5, byte2:=16#3B, byte3:=2, energy=>MB_vars.M11T2,done=>get_energy_M11T2_done);
		IF get_energy_M11T2_done = TRUE THEN
			Mercury.M11T2:=MB_vars.M11T2;
			state:=36;
		ELSIF tmcheck.Q THEN state:=888;
		END_IF
36:
		tmCheck(in:=FALSE);
		tmCheck(in:=TRUE,pt:=t#2s);
		get_energy_M12T1_done := FALSE;
		get_energy_M12T1(byte1:=5, byte2:=16#3C, byte3:=1,  energy=>MB_vars.M12T1, done=>get_energy_M12T1_done);
		IF get_energy_M12T1_done = TRUE THEN
			Mercury.M12T1:=MB_vars.M12T1;
			state:=37;
		ELSIF tmcheck.Q THEN state:=888;
		END_IF
37:
		tmCheck(in:=FALSE);
		tmCheck(in:=TRUE,pt:=t#2s);
		get_energy_M12T2_done := FALSE;
		get_energy_M12T2(byte1:=5, byte2:=16#3C, byte3:=2,  energy=>MB_vars.M12T2,done=>get_energy_M12T2_done);
		IF get_energy_M12T2_done = TRUE THEN
			Mercury.M12T2:=MB_vars.M12T2;
			state:=888;
		ELSIF tmcheck.Q THEN state:=888;
		END_IF



888:
		Timer1(IN:=NOT Timer1Q , PT:=T#60s , Q=>Timer1Q , ET=> );
		IF timer1.q THEN

		state:=0;
		END_IF

END_CASE

FtrigBusy(CLK:=mb.BUSY );
IF FtrigBusy.Q THEN
	IF mb.Error THEN
		LastModbusError := mb.ErrorDiagnostics;
		LastErrorstate := state;
		CounterError := CounterError + 1;
	ELSE
		CounterSuccess := CounterSuccess + 1;
	END_IF
END_IF



SerialLinecontrolCom1(
	mode:=SerialLinemode_kl6_22b_standard,
	pComIn:=ADR(RS485read.MB.InData),
	pComOut:=ADR(RS485read.MB.OutData),
	SizeComIn:=SIZEOF(RS485read.MB.OutData),
	TxBuffer:=TxBufferCom1,
	RxBuffer:=RxBufferCom1,
	Error=>,
	errorid=>);
END_PROGRAM

(* POU FB_GET_CO2_MH_Z19B, ST *)
FUNCTION_BLOCK FB_GET_CO2_MH_Z19B
VAR_INPUT

END_VAR

VAR_OUTPUT
	co2				: REAL;
	done			: BOOL;
END_VAR

VAR
	SendBuffer		: ARRAY[0..8] OF BYTE;
	ReceiveBuffer	: ARRAY[0..13] OF BYTE;
	Clear			: ClearComBuffer;
	state			: INT:= 0;
	tmcheck			: TON;
	w_CO2		:	WORD;
END_VAR
tmcheck();

CASE state OF

0:
	done:=FALSE;
	Clear(Buffer := RxBufferCom1);
	SendBuffer[0] := 16#FF;
	SendBuffer[1] := 16#01; (* Address *)
	SendBuffer[2] := 16#86;
	SendBuffer[3] := 16#00;
	SendBuffer[4] := 16#00;
	SendBuffer[5] := 16#00;
	SendBuffer[6] := 16#00;
	SendBuffer[7] := 16#00;	(* Checksum *)
	SendBuffer[8] := 16#79;	(* Checksum *)

	SendDataCom1(pSendData:=ADR(SendBuffer),length:=9,TXbuffer:=TXBufferCom1,Busy=>,Error=>);

	tmCheck(in:=FALSE);
	tmCheck(in:=TRUE,pt:=t#2s);
	state:=1;

1: (*ответ*)

	ReceiveDataCom1(pPrefix:=,LenPrefix:=,pSuffix:=,LenSuffix:=,pReceiveData:=ADR(ReceiveBuffer),SizeReceiveData:=9,TImeOut:=t#1s,Reset:=,RXbuffer:=RxBufferCom1,DataReceived=>,busy=>,RxTimeout=>,LenReceiveData=>);

	IF ReceiveDataCom1.Error <> 0 THEN
		state:=9;
	END_IF

	IF ReceiveDataCom1.DataReceived THEN
		state:=2;
	ELSIF tmcheck.Q THEN
		 state:=9;
	END_IF;



2:(*расшифровка*)
	IF (ReceiveBuffer [0] = 16#FF AND ReceiveBuffer [1] = 16#86 ) THEN
		Sensor_CO2_high := ReceiveBuffer [2];
		Sensor_CO2_low := ReceiveBuffer [3];
		MEMCPY(ADR(w_CO2),ADR(ReceiveBuffer[3]),1);
		MEMCPY(ADR(w_CO2)+1,ADR(ReceiveBuffer[2]),1);
		IF (WORD_TO_REAL(w_CO2)<>0 AND WORD_TO_REAL(w_CO2)<5001) THEN
			co2 := WORD_TO_REAL(w_CO2);
			state:=10;
		ELSE
			state:=9;
		END_IF
	ELSE
		state:=9;
	END_IF

9:
	co2:=0;
	done := TRUE;
	state:=0;
10:
	done := TRUE;
	state:=0;

END_CASE;
END_FUNCTION_BLOCK

(* POU FB_GET_SUPPLY, ST *)
FUNCTION_BLOCK FB_GET_SUPPLY
VAR_INPUT
	byte1			: BYTE;
	byte2			: BYTE;
	byte3			: BYTE;

END_VAR

VAR_OUTPUT
	supply1			: REAL;
	supply2			: REAL;
	supply3			: REAL;
	done			: BOOL;
END_VAR

VAR

	Clear			: ClearComBuffer;
	crctest			: WORD;
	arrReceive		: ARRAY[1..12] OF BYTE := 0,0,0,0,0,0,0,0,0,0,0,0;
	arrSend			: ARRAY[1..6] OF BYTE:= 0,0,0,0,0,0;
	state			: INT:= 0;
	dw_DATA		: DWORD:=0;
	tmcheck			: TON;
	CRC_calc		: WORD:=0;
	CRC_get			: WORD:=1;

END_VAR
tmcheck();

CASE state OF

0:

	done:=FALSE;
	Clear(Buffer := RxBufferCom1);

	arrSend[1]:=Merc_address;
	arrSend[2]:=byte1;
	arrSend[3]:=byte2;
	arrSend[4]:=byte3;

	crctest:=F_CRC16(ADR(arrSend), 4);
	MEMCPY(ADR(arrSend)+4,ADR(crctest),2);

	SendDataCom1(pSendData:=ADR(arrSend),length:=6,TXbuffer:=TXBufferCom1 );

	tmCheck(in:=FALSE);
	tmCheck(in:=TRUE,pt:=t#2s);
	state:=1;

1: (*ответ*)

	ReceiveDataCom1(pReceiveData:=ADR(arrReceive),SizeReceiveData:=12,TImeOut:=t#2s,Reset:=,RXbuffer:=RxBufferCom1);

	IF ReceiveDataCom1.Error <> 0 THEN
		state:=9;
	END_IF

	IF ReceiveDataCom1.DataReceived THEN
		state:=2;

	ELSIF tmcheck.Q THEN state:=9;
	END_IF;


2:(*расшифровка*)
	(* arrReceive:=EchoDel(CheckUp:=TRUE, SentA:=arrSend, RecA:=arrReceive, Length:=UDINT_TO_INT(SendDataCom1.Length)); *)
	CRC_calc := F_CRC16(ADR(arrReceive), 10);
	MEMCPY(ADR(CRC_get),ADR(arrReceive[11]),1);
	MEMCPY(ADR(CRC_get)+1,ADR(arrReceive[12]),1);


	IF (  arrReceive[1] = Merc_address  AND CRC_calc = CRC_get ) THEN
		MEMCPY(ADR(dw_DATA),ADR(arrReceive[3]),1);
			MEMCPY(ADR(dw_DATA)+1,ADR(arrReceive[4]),1);
			arrReceive[2]:=arrReceive[2] AND 16#3F;
			MEMCPY(ADR(dw_DATA)+2,ADR(arrReceive[2]),1);
		supply1:=DWORD_TO_REAL(dw_DATA)/100;  (*Вольт*)

		MEMCPY(ADR(dw_DATA),ADR(arrReceive[6]),1);
			MEMCPY(ADR(dw_DATA)+1,ADR(arrReceive[7]),1);
			arrReceive[5]:=arrReceive[5] AND 16#3F;
			MEMCPY(ADR(dw_DATA)+2,ADR(arrReceive[5]),1);
		supply2:=DWORD_TO_REAL(dw_DATA)/100;  (*Вольт*)

		MEMCPY(ADR(dw_DATA),ADR(arrReceive[9]),1);
			MEMCPY(ADR(dw_DATA)+1,ADR(arrReceive[10]),1);
			arrReceive[8]:=arrReceive[8] AND 16#3F;
			MEMCPY(ADR(dw_DATA)+2,ADR(arrReceive[8]),1);
		supply3:=DWORD_TO_REAL(dw_DATA)/100;  (*Вольт*)



			state:=10;
		ELSE state:=9;
	END_IF;

9:
	supply1:=0;
	supply2:=0;
	supply3:=0;
	done := TRUE;
	state:=0;

10:
	done := TRUE;
	state:=0;

END_CASE;
END_FUNCTION_BLOCK

(* POU MB_func/F_CRC16, ST *)
FUNCTION F_CRC16 : WORD
VAR_INPUT
	pData: POINTER TO BYTE;		(* указатель на блок данных *)
	Size: WORD;						(* размер блока  данных *)
END_VAR
VAR
	Cnt: BYTE;							(* счетчик битов *)
END_VAR
F_CRC16 := 16#FFFF;
WHILE Size > 0 DO
	F_CRC16 := F_CRC16 XOR pData^;
	FOR Cnt := 0 TO 7 DO
		IF F_CRC16.0 = 0 THEN
			F_CRC16 := SHR(F_CRC16, 1);
		ELSE
			F_CRC16 := SHR(F_CRC16, 1) XOR 16#A001;
		END_IF
	END_FOR;
	pData := pData + 1;
	Size := Size - 1;
END_WHILE
END_FUNCTION

(* POU FB_GET_CURRENT, ST *)
FUNCTION_BLOCK FB_GET_CURRENT
VAR_INPUT
	byte1			: BYTE;
	byte2			: BYTE;
	byte3			: BYTE;

END_VAR

VAR_OUTPUT
	current1			: REAL;
	current2			: REAL;
	current3			: REAL;
	done			: BOOL;
END_VAR

VAR
	Clear			: ClearComBuffer;
	crctest			: WORD;
	arrReceive		: ARRAY[1..12] OF BYTE := 0,0,0,0,0,0,0,0,0,0,0,0;
	arrSend			: ARRAY[1..6] OF BYTE:= 0,0,0,0,0,0;
	state			: INT:= 0;
	dw_DATA		: DWORD:=0;
	tmcheck			: TON;
	CRC_calc		: WORD:=0;
	CRC_get			: WORD:=1;
END_VAR
tmcheck();

CASE state OF

0:
	done:=FALSE;
	Clear(Buffer := RxBufferCom1);
	arrSend[1]:=Merc_address;
	arrSend[2]:=byte1;
	arrSend[3]:=byte2;
	arrSend[4]:=byte3;

	crctest:=F_CRC16(ADR(arrSend), 4);
	MEMCPY(ADR(arrSend)+4,ADR(crctest),2);

	SendDataCom1(pSendData:=ADR(arrSend),length:=6,TXbuffer:=TXBufferCom1 );

	tmCheck(in:=FALSE);
	tmCheck(in:=TRUE,pt:=t#2s);
	state:=1;

1: (*ответ*)

	ReceiveDataCom1(pReceiveData:=ADR(arrReceive),SizeReceiveData:=12,TImeOut:=t#2s,Reset:=,RXbuffer:=RxBufferCom1);

	IF ReceiveDataCom1.Error <> 0 THEN
		state:=9;
	END_IF

	IF ReceiveDataCom1.DataReceived THEN
		state:=2;
	ELSIF tmcheck.Q THEN state:=9;
	END_IF;


2:(*расшифровка*)

	CRC_calc := F_CRC16(ADR(arrReceive), 10);
	MEMCPY(ADR(CRC_get),ADR(arrReceive[11]),1);
	MEMCPY(ADR(CRC_get)+1,ADR(arrReceive[12]),1);


	IF (  arrReceive[1] = Merc_address  AND CRC_calc = CRC_get ) THEN

			MEMCPY(ADR(dw_DATA),ADR(arrReceive[3]),1);
			MEMCPY(ADR(dw_DATA)+1,ADR(arrReceive[4]),1);
			arrReceive[2]:=arrReceive[2] AND 16#3F;
			MEMCPY(ADR(dw_DATA)+2,ADR(arrReceive[2]),1);
			current1 :=DWORD_TO_REAL(dw_DATA)/1000;  (*Ампер*)

			MEMCPY(ADR(dw_DATA),ADR(arrReceive[6]),1);
			MEMCPY(ADR(dw_DATA)+1,ADR(arrReceive[7]),1);
			arrReceive[5]:=arrReceive[5] AND 16#3F;
			MEMCPY(ADR(dw_DATA)+2,ADR(arrReceive[5]),1);
			current2:=DWORD_TO_REAL(dw_DATA)/1000;  (*Ампер*)

			MEMCPY(ADR(dw_DATA),ADR(arrReceive[9]),1);
			MEMCPY(ADR(dw_DATA)+1,ADR(arrReceive[10]),1);
			arrReceive[8]:=arrReceive[8] AND 16#3F;
			MEMCPY(ADR(dw_DATA)+2,ADR(arrReceive[8]),1);
			current3 :=DWORD_TO_REAL(dw_DATA)/1000;  (*Ампер*)
			state:=10;
		ELSE state:=9;
	END_IF;

9:
	current1:=0;
	current2:=0;
	current3:=0;
	done := TRUE;
	state:=0;
10:
	done := TRUE;
	state:=0;

END_CASE;
END_FUNCTION_BLOCK

(* POU FB_GET_POWER, ST *)
FUNCTION_BLOCK FB_GET_POWER
VAR_INPUT
	byte1			: BYTE;
	byte2			: BYTE;
	byte3			: BYTE;
END_VAR

VAR_OUTPUT
	power_total		: REAL;
	power1			: REAL;
	power2			: REAL;
	power3			: REAL;
	done			: BOOL;
END_VAR

VAR
	Clear				: ClearComBuffer;
	crctest				: WORD;
	arrReceive			: ARRAY[1..15] OF BYTE := 0,0,0,0,0,0,0,0,0,0,0,0,0,0,0;
	arrSend				: ARRAY[1..6] OF BYTE:= 0,0,0,0,0,0;
	state				: INT:= 0;
	dw_DATA			: DWORD:=0;
	tmcheck				: TON;
	CRC_calc			: WORD:=0;
	CRC_get				: WORD:=1;
END_VAR
tmcheck();

CASE state OF

0:
	done:=FALSE;
	Clear(Buffer := RxBufferCom1);
	arrSend[1]:=Merc_address;
	arrSend[2]:=byte1;
	arrSend[3]:=byte2;
	arrSend[4]:=byte3;

	crctest:=F_CRC16(ADR(arrSend), 4);
	MEMCPY(ADR(arrSend)+4,ADR(crctest),2);

	SendDataCom1(pSendData:=ADR(arrSend),length:=6,TXbuffer:=TXBufferCom1 );

	tmCheck(in:=FALSE);
	tmCheck(in:=TRUE,pt:=t#2s);
	state:=1;

1: (*ответ*)

	ReceiveDataCom1(pReceiveData:=ADR(arrReceive),SizeReceiveData:=15,TImeOut:=t#2s,Reset:=,RXbuffer:=RxBufferCom1);

	IF ReceiveDataCom1.Error <> 0 THEN
		state:=9;
	END_IF

	IF ReceiveDataCom1.DataReceived THEN
		state:=2;
	ELSIF tmcheck.Q THEN state:=9;
	END_IF;


2:(*расшифровка*)
	CRC_calc := F_CRC16(ADR(arrReceive), 13);
	MEMCPY(ADR(CRC_get),ADR(arrReceive[14]),1);
	MEMCPY(ADR(CRC_get)+1,ADR(arrReceive[15]),1);


	IF (  arrReceive[1] = Merc_address  AND CRC_calc = CRC_get ) THEN
			MEMCPY(ADR(dw_DATA),ADR(arrReceive[3]),1);
			MEMCPY(ADR(dw_DATA)+1,ADR(arrReceive[4]),1);
			arrReceive[2]:=arrReceive[2] AND 16#3F;
			MEMCPY(ADR(dw_DATA)+2,ADR(arrReceive[2]),1);
			power_total:=DWORD_TO_REAL(dw_DATA)/100;

			MEMCPY(ADR(dw_DATA),ADR(arrReceive[6]),1);
			MEMCPY(ADR(dw_DATA)+1,ADR(arrReceive[7]),1);
			arrReceive[5]:=arrReceive[5] AND 16#3F;
			MEMCPY(ADR(dw_DATA)+2,ADR(arrReceive[5]),1);
			power1:=DWORD_TO_REAL(dw_DATA)/100;

			MEMCPY(ADR(dw_DATA),ADR(arrReceive[9]),1);
			MEMCPY(ADR(dw_DATA)+1,ADR(arrReceive[10]),1);
			arrReceive[8]:=arrReceive[8] AND 16#3F;
			MEMCPY(ADR(dw_DATA)+2,ADR(arrReceive[8]),1);
			power2:=DWORD_TO_REAL(dw_DATA)/100;

			MEMCPY(ADR(dw_DATA),ADR(arrReceive[12]),1);
			MEMCPY(ADR(dw_DATA)+1,ADR(arrReceive[13]),1);
			arrReceive[11]:=arrReceive[11] AND 16#3F;
			MEMCPY(ADR(dw_DATA)+2,ADR(arrReceive[11]),1);
			power3:=DWORD_TO_REAL(dw_DATA)/100;



			state:=10;
		ELSE state:=9;
	END_IF;

9:
	power_total:=0;
	power1:=0;
	power2:=0;
	power3:=0;

	done := TRUE;
	state:=0;
10:
	done := TRUE;
	state:=0;

END_CASE;
END_FUNCTION_BLOCK

(* POU FB_GET_ENERGY, ST *)
FUNCTION_BLOCK FB_GET_ENERGY
VAR_INPUT
	byte1			: BYTE;
	byte2			: BYTE;
	byte3			: BYTE;
END_VAR

VAR_OUTPUT
	energy			: REAL;
	done			: BOOL;
END_VAR

VAR

	Clear				: ClearComBuffer;
	crctest				: WORD;
	arrReceive			: ARRAY[1..22] OF BYTE := 0,0,0,0,0,0,0,0,0,0,0,0,0,0,0,0,0,0,0,0,0,0;
	arrSend				: ARRAY[1..22] OF BYTE:= 0,0,0,0,0,0,0,0,0,0,0,0,0,0,0,0,0,0,0,0,0,0;
	state				: INT:= 0;
	dw_DATA			: DWORD:=0;
	E_active				: REAL:=0;
	E_reactive			: REAL:=0;
	tmcheck				: TON;
	CRC_calc			: WORD:=0;
	CRC_get				: WORD:=1;
END_VAR
tmcheck();

CASE state OF

0:
	done:=FALSE;
	Clear(Buffer := RxBufferCom1);
	arrSend[1]:=Merc_address;
	arrSend[2]:=byte1;
	arrSend[3]:=byte2;
	arrSend[4]:=byte3;

	crctest:=F_CRC16(ADR(arrSend), 4);
	MEMCPY(ADR(arrSend)+4,ADR(crctest),2);

	SendDataCom1(pSendData:=ADR(arrSend),length:=6,TXbuffer:=TXBufferCom1 );

	tmCheck(in:=FALSE);
	tmCheck(in:=TRUE,pt:=t#2s);
	state:=1;

1: (*ответ*)

	ReceiveDataCom1(pReceiveData:=ADR(arrReceive),SizeReceiveData:=19,TImeOut:=t#2s,Reset:=,RXbuffer:=RxBufferCom1);

	IF ReceiveDataCom1.Error <> 0 THEN
		state:=9;
	END_IF

	IF ReceiveDataCom1.DataReceived THEN
		state:=2;
	ELSIF tmcheck.Q THEN state:=9;
	END_IF;


2:(*расшифровка*)
	CRC_calc := F_CRC16(ADR(arrReceive), 17);
	MEMCPY(ADR(CRC_get),ADR(arrReceive[18]),1);
	MEMCPY(ADR(CRC_get)+1,ADR(arrReceive[19]),1);

	IF (  arrReceive[1] = Merc_address  AND CRC_calc = CRC_get ) THEN
			MEMCPY(ADR(dw_DATA),ADR(arrReceive[4]),2);
			MEMCPY(ADR(dw_DATA)+2,ADR(arrReceive[2]),2);
			E_active:=DWORD_TO_REAL(dw_DATA)/1000;(*активная мощ*)
			MEMCPY(ADR(dw_DATA),ADR(arrReceive[12]),2);
			MEMCPY(ADR(dw_DATA)+2,ADR(arrReceive[10]),2);
			E_reactive:=DWORD_TO_REAL(dw_DATA)/1000; (*реактивная мощность*)
			energy:=E_active;
			state:=10;
		ELSE state:=9;
	END_IF;
9:
	energy:=0;
	done := TRUE;
	state:=0;
10:
	done := TRUE;
	state:=0;

END_CASE;
END_FUNCTION_BLOCK

(* POU Mqtt, ST *)
PROGRAM Mqtt
VAR
	FB_Mqtt_Controller 		: FB_Mqtt_Controller_V10;
	stMqttSettings				: ST_MqttSettings;
	bMqttControllerBusy		: BOOL;

	FB_Mqtt_Publish1 			: FB_Mqtt_Publish_V10;
	FB_Mqtt_Publish2			: FB_Mqtt_Publish_V10;
	FB_Mqtt_Publish3			: FB_Mqtt_Publish_V10;
	FB_Mqtt_Publish4			: FB_Mqtt_Publish_V10;
	FB_Mqtt_Publish5			: FB_Mqtt_Publish_V10;
	FB_Mqtt_Publish6			: FB_Mqtt_Publish_V10;
	FB_Mqtt_Publish7			: FB_Mqtt_Publish_V10;
	FB_Mqtt_Publish8			: FB_Mqtt_Publish_V10;
	FB_Mqtt_Publish9			: FB_Mqtt_Publish_V10;
	FB_Mqtt_Publish10		: FB_Mqtt_Publish_V10;
	FB_Mqtt_Publish11		: FB_Mqtt_Publish_V10;
	FB_Mqtt_Publish12		: FB_Mqtt_Publish_V10;
	FB_Mqtt_Publish13 		: FB_Mqtt_Publish_V10;
	FB_Mqtt_Publish14		: FB_Mqtt_Publish_V10;
	FB_Mqtt_Publish15		: FB_Mqtt_Publish_V10;
	FB_Mqtt_Publish16		: FB_Mqtt_Publish_V10;
	FB_Mqtt_Publish17		: FB_Mqtt_Publish_V10;
	FB_Mqtt_Publish18		: FB_Mqtt_Publish_V10;
	FB_Mqtt_Publish19		: FB_Mqtt_Publish_V10;
	FB_Mqtt_Publish20		: FB_Mqtt_Publish_V10;
	FB_Mqtt_Publish21		: FB_Mqtt_Publish_V10;
	FB_Mqtt_Publish22		: FB_Mqtt_Publish_V10;
	FB_Mqtt_Publish23		: FB_Mqtt_Publish_V10;
	FB_Mqtt_Publish24		: FB_Mqtt_Publish_V10;

	bPublishBusy1			: BOOL;
	bPublishBusy2			: BOOL;
	bPublishBusy3			: BOOL;
	bPublishBusy4			: BOOL;
	bPublishBusy5			: BOOL;
	bPublishBusy6			: BOOL;
	bPublishBusy7			: BOOL;
	bPublishBusy8			: BOOL;
	bPublishBusy9			: BOOL;
	bPublishBusy10			: BOOL;
	bPublishBusy11			: BOOL;
	bPublishBusy12			: BOOL;
	bPublishBusy13			: BOOL;
	bPublishBusy14			: BOOL;
	bPublishBusy15			: BOOL;
	bPublishBusy16			: BOOL;
	bPublishBusy17			: BOOL;
	bPublishBusy18			: BOOL;
	bPublishBusy19			: BOOL;
	bPublishBusy20			: BOOL;
	bPublishBusy21			: BOOL;
	bPublishBusy22			: BOOL;
	bPublishBusy23			: BOOL;
	bPublishBusy24			: BOOL;
	START: BOOL;
END_VAR
FB_Mqtt_Controller (
		bActive			:= TRUE,
		sMqttClientId		:= 'plc',
		sMqttUserId		:= 'mqtt',
		sMqttPassword	:= 'mqtt',
		sMqttBrokerIp		:= '192.168.2.200',
		nMqttBrokerPort	:= 1883,
		stMqttSettings		:= stMqttSettings,
		bBusy			=> bMqttControllerBusy
	);

IF NOT bMqttControllerBusy THEN

	FB_Mqtt_Publish1(sTopic:='BECKHOFF_CX9000/Mercury/M1T1',sValue:=REAL_TO_STRING(Mercury.M1T1),bRetain:=FALSE, stMqttSettings:=stMqttSettings,bBusy => bPublishBusy1 );
	FB_Mqtt_Publish2(sTopic:='BECKHOFF_CX9000/Mercury/M1T2',sValue:=REAL_TO_STRING(Mercury.M1T2),bRetain:=FALSE, stMqttSettings:=stMqttSettings,bBusy => bPublishBusy2 );
	FB_Mqtt_Publish3(sTopic:='BECKHOFF_CX9000/Mercury/M2T1',sValue:=REAL_TO_STRING(Mercury.M2T1),bRetain:=FALSE, stMqttSettings:=stMqttSettings,bBusy => bPublishBusy3 );
	FB_Mqtt_Publish4(sTopic:='BECKHOFF_CX9000/Mercury/M2T2',sValue:=REAL_TO_STRING(Mercury.M2T2),bRetain:=FALSE, stMqttSettings:=stMqttSettings,bBusy => bPublishBusy4 );
	FB_Mqtt_Publish5(sTopic:='BECKHOFF_CX9000/Mercury/M3T1',sValue:=REAL_TO_STRING(Mercury.M3T1),bRetain:=FALSE, stMqttSettings:=stMqttSettings,bBusy => bPublishBusy5 );
	FB_Mqtt_Publish6(sTopic:='BECKHOFF_CX9000/Mercury/M3T2',sValue:=REAL_TO_STRING(Mercury.M3T2),bRetain:=FALSE, stMqttSettings:=stMqttSettings,bBusy => bPublishBusy6 );
	FB_Mqtt_Publish7(sTopic:='BECKHOFF_CX9000/Mercury/M4T1',sValue:=REAL_TO_STRING(Mercury.M4T1),bRetain:=FALSE, stMqttSettings:=stMqttSettings,bBusy => bPublishBusy7 );
	FB_Mqtt_Publish8(sTopic:='BECKHOFF_CX9000/Mercury/M4T2',sValue:=REAL_TO_STRING(Mercury.M4T2),bRetain:=FALSE, stMqttSettings:=stMqttSettings,bBusy => bPublishBusy8 );
	FB_Mqtt_Publish9(sTopic:='BECKHOFF_CX9000/Mercury/M5T1',sValue:=REAL_TO_STRING(Mercury.M5T1),bRetain:=FALSE, stMqttSettings:=stMqttSettings,bBusy => bPublishBusy9 );
	FB_Mqtt_Publish10(sTopic:='BECKHOFF_CX9000/Mercury/M5T2',sValue:=REAL_TO_STRING(Mercury.M5T2),bRetain:=FALSE, stMqttSettings:=stMqttSettings,bBusy => bPublishBusy10 );
	FB_Mqtt_Publish11(sTopic:='BECKHOFF_CX9000/Mercury/M6T1',sValue:=REAL_TO_STRING(Mercury.M6T1),bRetain:=FALSE, stMqttSettings:=stMqttSettings,bBusy => bPublishBusy11 );
	FB_Mqtt_Publish12(sTopic:='BECKHOFF_CX9000/Mercury/M6T2',sValue:=REAL_TO_STRING(Mercury.M6T2),bRetain:=FALSE, stMqttSettings:=stMqttSettings,bBusy => bPublishBusy12 );
	FB_Mqtt_Publish13(sTopic:='BECKHOFF_CX9000/Mercury/M7T1',sValue:=REAL_TO_STRING(Mercury.M7T1),bRetain:=FALSE, stMqttSettings:=stMqttSettings,bBusy => bPublishBusy13 );
	FB_Mqtt_Publish14(sTopic:='BECKHOFF_CX9000/Mercury/M7T2',sValue:=REAL_TO_STRING(Mercury.M7T2),bRetain:=FALSE, stMqttSettings:=stMqttSettings,bBusy => bPublishBusy14);
	FB_Mqtt_Publish15(sTopic:='BECKHOFF_CX9000/Mercury/M8T1',sValue:=REAL_TO_STRING(Mercury.M8T1),bRetain:=FALSE, stMqttSettings:=stMqttSettings,bBusy => bPublishBusy15 );
	FB_Mqtt_Publish16(sTopic:='BECKHOFF_CX9000/Mercury/M8T2',sValue:=REAL_TO_STRING(Mercury.M8T2),bRetain:=FALSE, stMqttSettings:=stMqttSettings,bBusy => bPublishBusy16 );
	FB_Mqtt_Publish17(sTopic:='BECKHOFF_CX9000/Mercury/M9T1',sValue:=REAL_TO_STRING(Mercury.M9T1),bRetain:=FALSE, stMqttSettings:=stMqttSettings,bBusy => bPublishBusy17 );
	FB_Mqtt_Publish18(sTopic:='BECKHOFF_CX9000/Mercury/M9T2',sValue:=REAL_TO_STRING(Mercury.M9T2),bRetain:=FALSE, stMqttSettings:=stMqttSettings,bBusy => bPublishBusy18 );
	FB_Mqtt_Publish19(sTopic:='BECKHOFF_CX9000/Mercury/M10T1',sValue:=REAL_TO_STRING(Mercury.M10T1),bRetain:=FALSE, stMqttSettings:=stMqttSettings,bBusy => bPublishBusy19 );
	FB_Mqtt_Publish20(sTopic:='BECKHOFF_CX9000/Mercury/M10T2',sValue:=REAL_TO_STRING(Mercury.M10T2),bRetain:=FALSE, stMqttSettings:=stMqttSettings,bBusy => bPublishBusy20 );
	FB_Mqtt_Publish21(sTopic:='BECKHOFF_CX9000/Mercury/M11T1',sValue:=REAL_TO_STRING(Mercury.M11T1),bRetain:=FALSE, stMqttSettings:=stMqttSettings,bBusy => bPublishBusy21 );
	FB_Mqtt_Publish22(sTopic:='BECKHOFF_CX9000/Mercury/M11T2',sValue:=REAL_TO_STRING(Mercury.M11T2),bRetain:=FALSE, stMqttSettings:=stMqttSettings,bBusy => bPublishBusy22 );
	FB_Mqtt_Publish23(sTopic:='BECKHOFF_CX9000/Mercury/M12T1',sValue:=REAL_TO_STRING(Mercury.M12T1),bRetain:=FALSE, stMqttSettings:=stMqttSettings,bBusy => bPublishBusy23 );
	FB_Mqtt_Publish24(sTopic:='BECKHOFF_CX9000/Mercury/M12T2',sValue:=REAL_TO_STRING(Mercury.M12T2),bRetain:=FALSE, stMqttSettings:=stMqttSettings,bBusy => bPublishBusy24 );
END_IF
(*    END    SEND DATA VIA MQTT  *)
END_PROGRAM

(* POU FB_Mqtt_Controller_V10, ST *)
(* @NESTEDCOMMENTS := 'Yes' *)
(* @PATH := '\/_Generic\/Mqtt' *)
(* @OBJECTFLAGS := '0, 8' *)
(* @SYMFILEFLAGS := '2048' *)
FUNCTION_BLOCK FB_Mqtt_Controller_V10
VAR_INPUT
(*	bActive			: BOOL := FALSE;
	sMqttClientId	: STRING[23]:='plc';
	sMqttUserId	: STRING[25] := 'mqtt';
	sMqttPassword	: STRING[25] := 'mqtt';
	sMqttBrokerIP	: STRING[15]:='192.168.3.200';
	nMqttBrokerPort	: UDINT := 1883;
*)
	bActive			: BOOL := FALSE;
	sMqttClientId	: STRING[23];
	sMqttUserId	: STRING[25] := '';
	sMqttPassword	: STRING[25] := '';
	sMqttBrokerIP	: STRING[15];
	nMqttBrokerPort	: UDINT := 1883;
END_VAR
VAR_OUTPUT
	bBusy	: BOOL := FALSE;
END_VAR
VAR_IN_OUT
	stMqttSettings	: ST_MqttSettings;
END_VAR
VAR
	iState			: INT := 0;
	fbSocketConnect	: FB_SocketConnect;
	fbSocketClose	: FB_SocketClose;

	fbMqttTelegramConnect	: FB_MqttTelegram_Connect_V10;
	fbMqttTelegramPingReq	: FB_MqttTelegram_PingReq_V10;
	fbMqttSend				: FB_Mqtt_Send_V10;
	fbMqttReceive			: FB_Mqtt_Receive_V10;
END_VAR
VAR CONSTANT
	C_STARTUP					: INT := 0;
	C_CONNECT					: INT := 100;
	C_CONNECT_WAIT				: INT := 110;
	C_CLOSE						: INT := 200;
	C_CLOSE_WAIT				: INT := 210;
	C_IDLE						: INT := 500;
END_VAR
(* @END_DECLARATION := '0' *)
(*
 * Connects to mqtt broker
 * Sends connect message
 * Sends ping(back)
 * Sends disconnect
 *)
CASE iState OF
	C_STARTUP:
		stMqttSettings.bConnected			:= FALSE;
		stMqttSettings.bConnectPackageSent	:= FALSE;
		stMqttSettings.bDisconnect			:= FALSE;
		stMqttSettings.bSocketConnection	:= FALSE;
		stMqttSettings.bError				:= FALSE;
		stMqttSettings.bValidConnection		:= FALSE;
		stMqttSettings.wPackageIdentifier	:= 1;
		stMqttSettings.bActive				:= bActive;
		stMqttSettings.hSocket				:= fbSocketConnect.hSocket;
		stMqttSettings.nMqttBrokerPort		:= nMqttBrokerPort;
		stMqttSettings.sMqttBrokerIP		:= sMqttBrokerIP;
		stMqttSettings.sMqttClientId		:= sMqttClientId;
		stMqttSettings.sMqttUserId		:= sMqttUserId;
		stMqttSettings.sMqttPassword		:= sMqttPassword;

		stMqttSettings.stMqttReceivedTelegram.nDataLength := 0;

		bBusy := FALSE;

		CallMqttBlocks();

		IF bActive THEN
			iState := C_CONNECT;
		END_IF;

	(* Start connection *)
	C_CONNECT:
		bBusy := TRUE;

		fbSocketConnect(
			bExecute	:= FALSE
		);

		fbSocketConnect(
			sSrvNetId	:= '',
			sRemoteHost	:= sMqttBrokerIP,
			nRemotePort	:= nMqttBrokerPort,
			bExecute	:= TRUE,
			tTimeout	:= USINT_TO_TIME(stMqttSettings.usKeepAliveTime) + t#10s
		);

		iState := C_CONNECT_WAIT;

	(* Wait till connected *)
	C_CONNECT_WAIT:
		fbSocketConnect(
			bExecute := FALSE
		);

		IF
			NOT fbSocketConnect.bBusy
			AND NOT fbSocketConnect.bError
		THEN
			iState 								:= C_IDLE;
			stMqttSettings.hSocket				:= fbSocketConnect.hSocket;
			stMqttSettings.bSocketConnection	:= TRUE;
		END_IF;

		IF fbSocketConnect.bError THEN
			iState := C_STARTUP;
		END_IF;

		IF NOT stMqttSettings.bActive THEN
			iState := C_STARTUP;
		END_IF;

	(* Close connection *)
	C_CLOSE:
		bBusy := TRUE;

		fbSocketClose(
			bExecute	:= TRUE,
			hSocket		:= stMqttSettings.hSocket
		);

		iState := C_CLOSE_WAIT;

	(* Wait close connection *)
	C_CLOSE_WAIT:
		fbSocketClose(
			bExecute := FALSE
		);

		IF
			NOT fbSocketClose.bBusy
			AND NOT fbSocketClose.bError
		THEN
			iState := C_STARTUP;
		END_IF;

		IF fbSocketClose.bError THEN
			iState := C_STARTUP;
		END_IF;

		IF NOT stMqttSettings.bActive THEN
			iState := C_STARTUP;
		END_IF;

	(* Idle *)
	C_IDLE:
		bBusy 					:= FALSE;
		stMqttSettings.bActive	:= bActive;

		stMqttSettings.bValidConnection :=
			NOT stMqttSettings.bError
			AND NOT stMqttSettings.bDisconnect
			AND stMqttSettings.bConnected
			AND stMqttSettings.bSocketConnection
			AND stMqttSettings.bActive;

		CallMqttBlocks();

		IF
			stMqttSettings.bDisconnect
			OR stMqttSettings.bError
			OR NOT stMqttSettings.bActive
		THEN
			IF
				stMqttSettings.bConnected
				OR stMqttSettings.bSocketConnection
			THEN
				(* TODO : send disconnect *)
				iState := C_CLOSE;
			ELSE
				iState := C_CLOSE;
			END_IF;
		END_IF;

	ELSE
		iState := C_STARTUP;
END_CASE;
(*	END_FUNCTION_BLOCK	*)
END_FUNCTION_BLOCK
ACTION CallMqttBlocks:
(*ACTION	CallMqttBlocks: *)
fbMqttReceive(
	stMqttSettings := stMqttSettings
);

fbMqttTelegramConnect(
	stMqttSettings := stMqttSettings
);

fbMqttTelegramPingReq(
	stMqttSettings := stMqttSettings
);

fbMqttSend(
	stMqttSettings := stMqttSettings
);

(* END_ACTION *)
END_ACTION

(* POU Intern/FB_MqttTelegram_Connect_V10, ST *)
(* @NESTEDCOMMENTS := 'Yes' *)
(* @PATH := '\/_Generic\/Mqtt\/Intern' *)
(* @OBJECTFLAGS := '0, 8' *)
(* @SYMFILEFLAGS := '2048' *)
FUNCTION_BLOCK FB_MqttTelegram_Connect_V10
VAR_IN_OUT
	stMqttSettings	: ST_MqttSettings;
END_VAR
VAR
	iState 				: INT := 0;
	idLength			: INT;
	iuLength			: INT;
	ipLength			: INT;
	ipos				: INT;
	stMqttTelegram		: ST_MqttTelegram;
	fbMqttEncodeLength	: FB_Mqtt_EncodeLength_V10;
	bLength1			: BYTE;
	bLength2			: BYTE;
	bLength3			: BYTE;
	bLength4			: BYTE;
	bLengthAmount		: BYTE;
END_VAR
VAR CONSTANT
	C_STARTUP		: INT := 0;
	C_BUILD_CONNECT	: INT := 100;
	C_SEND_WAIT		: INT := 110;
	C_IDLE			: INT := 500;
END_VAR
(* @END_DECLARATION := '0' *)
CASE iState OF
	C_STARTUP:
		IF
			NOT stMqttSettings.bDisconnect
			AND NOT stMqttSettings.bError
			AND stMqttSettings.bSocketConnection
			AND stMqttSettings.bActive
		THEN
			iState := C_IDLE;
		END_IF;

	(* build connect telegram *)
	C_BUILD_CONNECT:
		FC_Mqtt_ClearTelegram_V10(
			stMqttTelegram	:= stMqttTelegram,
			stMqttSettings	:= stMqttSettings
		);

		(* get client id length *)
		idLength := LEN(stMqttSettings.sMqttClientId);
		IF idLength < 1 THEN
			stMqttSettings.sMqttClientId := 'x';
			idLength := 1;
		END_IF;

		IF idLength > 23 THEN
			idLength := 23;
		END_IF;

		IF
			LEN(stMqttSettings.sMqttUserId) > 0
			AND LEN(stMqttSettings.sMqttPassword) > 0
		THEN
			iuLength := LEN(stMqttSettings.sMqttUserId)+2; (* 2 byte data length*)
			ipLength := LEN(stMqttSettings.sMqttPassword)+2; (* 2 byte data length*)
		ELSE
			iuLength := 0;
			ipLength := 0;
		END_IF

		(* Calculate length *)
		(* 10 byte header, 2 byte data length, data length, [user length + 2], [password length + 2]*)
		fbMqttEncodeLength(
			dwLength := 10 + 2 + INT_TO_BYTE(idLength) + INT_TO_BYTE(iuLength) + INT_TO_BYTE(ipLength),
			bLength1 => bLength1,
			bLength2 => bLength2,
			bLength3 => bLength3,
			bLength4 => bLength4,
			bAmount	 => bLengthAmount
		);

		(* MQTT Control Packet type *)
		stMqttTelegram.arMqttData[0] := 16;
		(* Remaining Length *)
		CASE bLengthAmount OF
			1:
				stMqttTelegram.arMqttData[1] := bLength1;

			2:
				stMqttTelegram.arMqttData[1] := bLength1;
				stMqttTelegram.arMqttData[2] := bLength2;

			3:
				stMqttTelegram.arMqttData[1] := bLength1;
				stMqttTelegram.arMqttData[2] := bLength2;
				stMqttTelegram.arMqttData[3] := bLength3;

			4:
				stMqttTelegram.arMqttData[1] := bLength1;
				stMqttTelegram.arMqttData[2] := bLength2;
				stMqttTelegram.arMqttData[3] := bLength3;
				stMqttTelegram.arMqttData[4] := bLength4;
		END_CASE;
		(* init position*)
		ipos := bLengthAmount;

		(* Length MSB *)
		stMqttTelegram.arMqttData[ipos+1] := 0;
		(* Length LSB *)
		stMqttTelegram.arMqttData[ipos+2] := 4;
		(* M *)
		stMqttTelegram.arMqttData[ipos+3] := 77;
		(* Q *)
		stMqttTelegram.arMqttData[ipos+4] := 81;
		(* T *)
		stMqttTelegram.arMqttData[ipos+5] := 84;
		(* T *)
		stMqttTelegram.arMqttData[ipos+6] := 84;
		(* Protocol Level *)
		stMqttTelegram.arMqttData[ipos+7] := 4;
		(* Connect Flags *)
		stMqttTelegram.arMqttData[ipos+8].1 := TRUE;
		stMqttTelegram.arMqttData[ipos+8].6 := (ipLength>2); (* more then 2 byte data length*)
		stMqttTelegram.arMqttData[ipos+8].7 := (iuLength>2); (* more then 2 byte data length*)
		(* Keep Alive MSB *)
		stMqttTelegram.arMqttData[ipos+9] := 0;
		(* Keep Alive LSB *)
		stMqttTelegram.arMqttData[ipos+10] := stMqttSettings.usKeepAliveTime;
		(* Data length MSB *)
		stMqttTelegram.arMqttData[ipos+11] := 0;
		(* Data length LSB *)
		stMqttTelegram.arMqttData[ipos+12] := INT_TO_BYTE(idLength);

		(* Client ID *)
		MEMCPY(
			destAddr	:= ADR(stMqttTelegram.arMqttData[ipos+13]),
		    srcAddr		:= ADR(stMqttSettings.sMqttClientId),
			n  			:= idLength
		);

		ipos := ipos+13+idLength;
		IF (iuLength > 2) THEN (* more then 2 byte data length*)
			(* Data length MSB *)
			stMqttTelegram.arMqttData[ipos] := 0;
			(* Data length LSB *)
			stMqttTelegram.arMqttData[ipos+1] := INT_TO_BYTE(iuLength-2);

			(* User ID *)
			MEMCPY(
				destAddr	:= ADR(stMqttTelegram.arMqttData[ipos+2]),
			    srcAddr		:= ADR(stMqttSettings.sMqttUserId),
				n  			:= iuLength-2
			);
			ipos := ipos+iuLength;
		END_IF

		IF (iuLength > 2) THEN (* more then 2 byte data length*)
			(* Data length MSB *)
			stMqttTelegram.arMqttData[ipos] := 0;
			(* Data length LSB *)
			stMqttTelegram.arMqttData[ipos+1] := INT_TO_BYTE(ipLength-2);

			(* Password *)
			MEMCPY(
				destAddr	:= ADR(stMqttTelegram.arMqttData[ipos+2]),
			    srcAddr		:= ADR(stMqttSettings.sMqttPassword),
				n  			:= ipLength-2
			);
			ipos := ipos+ipLength;
		END_IF

		stMqttTelegram.nDataLength 	:= ipos; (* 1 byte header, 1 byte remaining length *)
		iState 						:= C_SEND_WAIT;

	(* send telegram *)
	C_SEND_WAIT:
		IF stMqttSettings.stMqttSendTelegram.nDataLength = 0 THEN
			FC_Mqtt_CopyTelegram_V10(
				stMqttSrcTelegram	:= stMqttTelegram,
				stMqttDestTelegram	:= stMqttSettings.stMqttSendTelegram,
				stMqttSettings		:= stMqttSettings
			);

			stMqttSettings.bConnectPackageSent	:= TRUE;
			iState								:= C_IDLE;
		END_IF;

		IF
			NOT stMqttSettings.bActive
			OR NOT stMqttSettings.bSocketConnection
		THEN
			iState := C_STARTUP;
		END_IF;

	(* idle *)
	C_IDLE:
		IF
			NOT stMqttSettings.bDisconnect
			AND NOT stMqttSettings.bError
			AND NOT stMqttSettings.bConnected
			AND stMqttSettings.bSocketConnection
			AND NOT stMqttSettings.bConnectPackageSent
			AND stMqttSettings.bActive
		THEN
			iState := C_BUILD_CONNECT;
		END_IF;

		(* check received telegram *)
		IF
			stMqttSettings.bConnectPackageSent
			AND stMqttSettings.stMqttReceivedTelegram.nDataLength = 4
			AND stMqttSettings.stMqttReceivedTelegram.arMqttData[0] = 32
			AND stMqttSettings.stMqttReceivedTelegram.arMqttData[1] = 2
			AND (
				(* Session pressent or not, we ignore *)
				stMqttSettings.stMqttReceivedTelegram.arMqttData[2] = 1
				OR
				stMqttSettings.stMqttReceivedTelegram.arMqttData[2] = 0
			)
			AND stMqttSettings.stMqttReceivedTelegram.arMqttData[3] = 0
		THEN
			stMqttSettings.bConnected := TRUE;
			FC_Mqtt_ClearTelegram_V10(
				stMqttTelegram	:= stMqttSettings.stMqttReceivedTelegram,
				stMqttSettings	:= stMqttSettings
			);
		END_IF;

		(* error on connect *)
		IF
			stMqttSettings.bConnectPackageSent
			AND stMqttSettings.stMqttReceivedTelegram.nDataLength = 4
			AND stMqttSettings.stMqttReceivedTelegram.arMqttData[0] = 32
			AND stMqttSettings.stMqttReceivedTelegram.arMqttData[1] = 2
			AND stMqttSettings.stMqttReceivedTelegram.arMqttData[3] <> 0
		THEN
			stMqttSettings.bError := TRUE;
		END_IF;

		IF
			stMqttSettings.bDisconnect
			OR stMqttSettings.bError
			OR NOT stMqttSettings.bSocketConnection
			OR NOT stMqttSettings.bActive
		THEN
			iState := C_STARTUP;
		END_IF;

	ELSE
		iState := C_STARTUP;
END_CASE;


(*	END_FUNCTION_BLOCK	*)
END_FUNCTION_BLOCK

(* POU Intern/FB_Mqtt_EncodeLength_V10, ST *)
(* @NESTEDCOMMENTS := 'Yes' *)
(* @PATH := '\/_Generic\/Mqtt\/Intern' *)
(* @OBJECTFLAGS := '0, 8' *)
(* @SYMFILEFLAGS := '2048' *)
FUNCTION_BLOCK FB_Mqtt_EncodeLength_V10
VAR_INPUT
	dwLength	: DWORD;
END_VAR
VAR_OUTPUT
	bLength1	: BYTE := 0;
	bLength2	: BYTE := 0;
	bLength3	: BYTE := 0;
	bLength4	: BYTE := 0;
	bAmount		: BYTE := 0;
END_VAR
VAR
	dwWorkLength	: DWORD;
	dwCopyLength	: DWORD;
END_VAR
(* @END_DECLARATION := '0' *)
bAmount 		:= 1;
dwCopyLength	:= dwLength;

WHILE dwCopyLength > 0 DO
	dwWorkLength := dwCopyLength MOD 128;
	dwCopyLength := dwCopyLength / 128;

	IF dwCopyLength > 0 THEN
		dwWorkLength := dwWorkLength OR 128;
	END_IF;

	CASE bAmount OF
		1:
			bLength1 := DWORD_TO_BYTE(dwWorkLength);

		2:
			bLength2 := DWORD_TO_BYTE(dwWorkLength);

		3:
			bLength3 := DWORD_TO_BYTE(dwWorkLength);

		4:
			bLength4 := DWORD_TO_BYTE(dwWorkLength);

		ELSE
			;
	END_CASE;

	IF dwCopyLength > 0 THEN
		bAmount := bAmount + 1;
	END_IF;

	IF bAmount > 4 THEN
		(* hmm *)
		RETURN;
	END_IF;
END_WHILE;
(*
do
	encodedByte = X MOD 128
	X = X DIV 128

	// if there are more data to encode, set the top bit of this byte
	if ( X > 0 )
		encodedByte = encodedByte OR 128
	endif

	'output' encodedByte
while ( X > 0 )
*)

(*	END_FUNCTION_BLOCK	*)
END_FUNCTION_BLOCK

(* POU Intern/FC_Mqtt_ClearTelegram_V10, ST *)
(* @NESTEDCOMMENTS := 'Yes' *)
(* @PATH := '\/_Generic\/Mqtt\/Intern' *)
(* @OBJECTFLAGS := '0, 8' *)
(* @SYMFILEFLAGS := '2048' *)
FUNCTION FC_Mqtt_ClearTelegram_V10 : BOOL
VAR_IN_OUT
	stMqttTelegram	: ST_MqttTelegram;
	stMqttSettings	: ST_MqttSettings;
END_VAR
VAR
END_VAR
(* @END_DECLARATION := '0' *)
MEMSET(
	destAddr	:= ADR(stMqttTelegram.arMqttData),
	fillByte  	:= 0,
	n			:= stMqttSettings.iTelegramSize
);

stMqttTelegram.nDataLength := 0;

(*	END_FUNCTION	*)
END_FUNCTION

(* POU Intern/FC_Mqtt_CopyTelegram_V10, ST *)
(* @NESTEDCOMMENTS := 'Yes' *)
(* @PATH := '\/_Generic\/Mqtt\/Intern' *)
(* @OBJECTFLAGS := '0, 8' *)
(* @SYMFILEFLAGS := '2048' *)
FUNCTION FC_Mqtt_CopyTelegram_V10 : BOOL
VAR_IN_OUT
	stMqttSrcTelegram	: ST_MqttTelegram;
	stMqttDestTelegram	: ST_MqttTelegram;
	stMqttSettings		: ST_MqttSettings;
END_VAR
VAR
END_VAR
(* @END_DECLARATION := '0' *)
MEMCPY(
	destAddr	:= ADR(stMqttDestTelegram.arMqttData),
    srcAddr		:= ADR(stMqttSrcTelegram.arMqttData),
	n  			:= stMqttSettings.iTelegramSize
);

stMqttDestTelegram.nDataLength := stMqttSrcTelegram.nDataLength;

(*	END_FUNCTION	*)
END_FUNCTION

(* POU Intern/FB_MqttTelegram_PingReq_V10, ST *)
(* @NESTEDCOMMENTS := 'Yes' *)
(* @PATH := '\/_Generic\/Mqtt\/Intern' *)
(* @OBJECTFLAGS := '0, 8' *)
(* @SYMFILEFLAGS := '2048' *)
FUNCTION_BLOCK FB_MqttTelegram_PingReq_V10
VAR_IN_OUT
	stMqttSettings	: ST_MqttSettings;
END_VAR
VAR
	iState 				: INT := 0;
	bMustSend			: BOOL := FALSE;
	bPingReqSent		: BOOL := FALSE;
	stMqttTelegram		: ST_MqttTelegram;
END_VAR
VAR CONSTANT
	C_STARTUP		: INT := 0;
	C_BUILD_PING	: INT := 100;
	C_SEND_WAIT		: INT := 110;
	C_IDLE			: INT := 500;
END_VAR
(* @END_DECLARATION := '0' *)
CASE iState OF
	C_STARTUP:
		bPingReqSent := FALSE;

		IF stMqttSettings.bValidConnection THEN
			iState := C_IDLE;
		END_IF;

	(* build pingreq telegram *)
	C_BUILD_PING:
		FC_Mqtt_ClearTelegram_V10(
			stMqttTelegram	:= stMqttTelegram,
			stMqttSettings	:= stMqttSettings
		);

		(* MQTT Control Packet type *)
		stMqttTelegram.arMqttData[0] := 192;
		(* Remaining Length *)
		stMqttTelegram.arMqttData[1] := 0;

		stMqttTelegram.nDataLength := 2;

		iState := C_SEND_WAIT;

	(* send telegram *)
	C_SEND_WAIT:
		IF stMqttSettings.stMqttSendTelegram.nDataLength = 0 THEN
			FC_Mqtt_CopyTelegram_V10(
				stMqttSrcTelegram	:= stMqttTelegram,
				stMqttDestTelegram	:= stMqttSettings.stMqttSendTelegram,
				stMqttSettings		:= stMqttSettings
			);

			bPingReqSent	:= TRUE;
			iState			:= C_IDLE;
		END_IF;

		IF NOT stMqttSettings.bValidConnection THEN
			iState := C_STARTUP;
		END_IF;

	(* idle *)
	C_IDLE:
		bMustSend := FALSE;

		IF stMqttSettings.usKeepAliveTime > 0 THEN
			bMustSend := stMqttSettings.tonSendPingReq.Q;
		END_IF;

		IF
			stMqttSettings.bValidConnection
			AND bMustSend
			AND NOT bPingReqSent
		THEN
			iState := C_BUILD_PING;
		END_IF;

		(* Check received telegram *)
		IF
			bPingReqSent
			AND stMqttSettings.stMqttReceivedTelegram.nDataLength = 2
			AND stMqttSettings.stMqttReceivedTelegram.arMqttData[0] = 208
			AND stMqttSettings.stMqttReceivedTelegram.arMqttData[1] = 0
		THEN
			FC_Mqtt_ClearTelegram_V10(
				stMqttTelegram	:= stMqttSettings.stMqttReceivedTelegram,
				stMqttSettings	:= stMqttSettings
			);
			bPingReqSent := FALSE;
		END_IF;

		IF NOT stMqttSettings.bValidConnection THEN
			iState := C_STARTUP;
		END_IF;

	ELSE
		iState := C_STARTUP;
END_CASE;

(*	END_FUNCTION_BLOCK	*)
END_FUNCTION_BLOCK

(* POU Intern/FB_Mqtt_Send_V10, ST *)
(* @NESTEDCOMMENTS := 'Yes' *)
(* @PATH := '\/_Generic\/Mqtt\/Intern' *)
(* @OBJECTFLAGS := '0, 8' *)
(* @SYMFILEFLAGS := '2048' *)
FUNCTION_BLOCK FB_Mqtt_Send_V10
VAR_OUTPUT
	bBusy	: BOOL := FALSE;
END_VAR
VAR_IN_OUT
	stMqttSettings	: ST_MqttSettings;
END_VAR
VAR
	fbSocketSend 	: FB_SocketSend;
	tPingReq		: TIME;
	iState 			: INT := 0;
	stSendTelegram	: ST_MqttTelegram;
END_VAR
VAR CONSTANT
	C_STARTUP		: INT := 0;
	C_SEND			: INT := 100;
	C_SEND_WAIT		: INT := 110;
	C_IDLE			: INT := 500;
END_VAR
(* @END_DECLARATION := '0' *)
CASE iState OF
	C_STARTUP:
		bBusy := FALSE;

		stMqttSettings.tonSendPingReq(
			in := FALSE
		);

		IF
			NOT stMqttSettings.bDisconnect
			AND NOT stMqttSettings.bError
			AND stMqttSettings.bSocketConnection
		THEN
			iState := C_IDLE;
		END_IF;

	(* send mqtt telegram *)
	C_SEND:
		bBusy := TRUE;

		(* copy send telegram *)
		FC_Mqtt_CopyTelegram_V10(
			stMqttSrcTelegram	:= stMqttSettings.stMqttSendTelegram,
			stMqttDestTelegram	:= stSendTelegram,
			stMqttSettings		:= stMqttSettings
		);

		(* start send *)
		fbSocketSend(
			bExecute := FALSE
		);

		fbSocketSend(
			sSrvNetId	:= '',
			hSocket		:= stMqttSettings.hSocket,
			cbLen		:= stSendTelegram.nDataLength,
			pSrc		:= ADR(stSendTelegram.arMqttData),
			bExecute 	:= TRUE
		);

		iState := C_SEND_WAIT;

	(* wait send done *)
	C_SEND_WAIT:
		fbSocketSend(
			bExecute := FALSE
		);

		IF
			NOT fbSocketSend.bBusy
			AND NOT fbSocketSend.bError
		THEN
			(* copy last telegram *)
			FC_Mqtt_CopyTelegram_V10(
				stMqttSrcTelegram	:= stMqttSettings.stMqttSendTelegram,
				stMqttDestTelegram	:= stMqttSettings.stMqttLastSendTelegram,
				stMqttSettings		:= stMqttSettings
			);

			(* clear send buffer *)
			FC_Mqtt_ClearTelegram_V10(
				stMqttTelegram 	:= stMqttSettings.stMqttSendTelegram,
				stMqttSettings	:= stMqttSettings
			);

			iState	:= C_IDLE;
			bBusy	:= FALSE;
		END_IF;

		IF stMqttSettings.usKeepAliveTime > 0 THEN
			tPingReq := DWORD_TO_TIME(USINT_TO_DWORD(stMqttSettings.usKeepAliveTime) * 1000 - 5000);

			stMqttSettings.tonSendPingReq(
				in := FALSE
			);

			stMqttSettings.tonSendPingReq(
				in := TRUE,
				pt := tPingReq
			);
		END_IF;

		IF fbSocketSend.bError THEN
			iState 					:= C_STARTUP;
			stMqttSettings.bError	:= TRUE;
		END_IF;

		IF
			NOT stMqttSettings.bActive
			OR NOT stMqttSettings.bSocketConnection
		THEN
			iState := C_STARTUP;
		END_IF;

	(* idle *)
	C_IDLE:
		IF stMqttSettings.usKeepAliveTime > 0 THEN
			stMqttSettings.tonSendPingReq(
				in := stMqttSettings.bConnected
			);
		ELSE
			stMqttSettings.tonSendPingReq(
				in := FALSE
			);
		END_IF;

		IF
			stMqttSettings.stMqttSendTelegram.nDataLength > 0
			AND NOT stMqttSettings.bDisconnect
			AND NOT stMqttSettings.bError
			AND stMqttSettings.bSocketConnection
			AND NOT bBusy
		THEN
			iState := C_SEND;
		END_IF;

		IF
			stMqttSettings.bDisconnect
			OR stMqttSettings.bError
			OR NOT stMqttSettings.bSocketConnection
		THEN
			iState := C_STARTUP;
		END_IF;

		(* ensure at least 1 cycle pause *)
		(* bBusy := FALSE; *)

	ELSE
		iState := C_STARTUP;
END_CASE;

(*	END_FUNCTION_BLOCK	*)
END_FUNCTION_BLOCK

(* POU Intern/FB_Mqtt_Receive_V10, ST *)
(* @NESTEDCOMMENTS := 'Yes' *)
(* @PATH := '\/_Generic\/Mqtt\/Intern' *)
(* @OBJECTFLAGS := '0, 8' *)
(* @SYMFILEFLAGS := '2048' *)
FUNCTION_BLOCK FB_Mqtt_Receive_V10
VAR_OUTPUT
	bBusy	: BOOL := FALSE;
END_VAR
VAR_IN_OUT
	stMqttSettings	: ST_MqttSettings;
END_VAR
VAR
	fbSocketReceive		: FB_SocketReceive;
	fbMqttDecodeLength	: FB_Mqtt_DecodeLength_V10;
	stReceiveBuffer		: ST_MqttTelegram;

	iState 			: INT := 0;
	iLengthPosition	: INT := 0;
	index			: INT := 0;
	dwDataLength	: DWORD := 0;
	wTopicLength	: WORD := 0;
	dwValueLength	: DWORD := 0;
END_VAR
VAR CONSTANT
	C_STARTUP				: INT := 0;
	C_RECEIVE_HEADER		: INT := 100;
	C_RECEIVE_HEADER_WAIT	: INT := 110;
	C_RECEIVE_LENGTH		: INT := 120;
	C_RECEIVE_LENGTH_WAIT	: INT := 130;
	C_RECEIVE_DATA			: INT := 200;
	C_RECEIVE_DATA_WAIT		: INT := 210;
	C_IDLE					: INT := 500;
END_VAR

(* @END_DECLARATION := '0' *)
CASE iState OF
	C_STARTUP:
		bBusy 			:= FALSE;
		iLengthPosition	:= 0;
		index			:= 0;
		dwDataLength	:= 0;
		wTopicLength	:= 0;
		dwValueLength	:= 0;
		ClearReceivedPublishTelegram();

		IF
			NOT stMqttSettings.bDisconnect
			AND NOT stMqttSettings.bError
			AND stMqttSettings.bSocketConnection
		THEN
			iState := C_IDLE;
		END_IF;

	(* start receive header *)
	C_RECEIVE_HEADER:
		bBusy := TRUE;
		ClearReceivedPublishTelegram();

		fbSocketReceive(
			bExecute := FALSE
		);

		fbSocketReceive(
			sSrvNetId	:= '',
			hSocket		:= stMqttSettings.hSocket,
			cbLen		:= 2,
			pDest		:= ADR(stReceiveBuffer.arMqttData),
			bExecute 	:= TRUE
		);

		iState := C_RECEIVE_HEADER_WAIT;

	(* wait for header with length *)
	C_RECEIVE_HEADER_WAIT:
		fbSocketReceive(
			bExecute := FALSE
		);

		IF
			NOT fbSocketReceive.bBusy
			AND NOT fbSocketReceive.bError
			AND fbSocketReceive.nRecBytes = 2
		THEN
			iLengthPosition	:= 0;
			stMqttSettings.stMqttReceivedTelegram.arMqttData[0] := stReceiveBuffer.arMqttData[0];
			stMqttSettings.stMqttReceivedTelegram.arMqttData[1] := stReceiveBuffer.arMqttData[1];

			IF stMqttSettings.stMqttReceivedTelegram.arMqttData[1].7 = 1 THEN
				(* payload longer then 127 byte *)
				iLengthPosition := iLengthPosition + 1;
				iState			:= C_RECEIVE_LENGTH;
			ELSE
				IF stMqttSettings.stMqttReceivedTelegram.arMqttData[1] = 0 THEN
					(* no payload received *)
					stMqttSettings.stMqttReceivedTelegram.nDataLength := 2;

					(* copy last telegram *)
					FC_Mqtt_CopyTelegram_V10(
						stMqttSrcTelegram	:= stMqttSettings.stMqttReceivedTelegram,
						stMqttDestTelegram	:= stMqttSettings.stMqttLastReceivedTelegram,
						stMqttSettings		:= stMqttSettings
					);

					iState	:= C_IDLE;
					bBusy 	:= FALSE;
				ELSE
					iState := C_RECEIVE_DATA;
				END_IF;
			END_IF;
		END_IF;

		IF fbSocketReceive.bError THEN
			iState 					:= C_STARTUP;
			stMqttSettings.bError	:= TRUE;
		END_IF;

		IF fbSocketReceive.nRecBytes = 0 THEN
			iState	:= C_IDLE;
			bBusy	:= FALSE;
		END_IF;

		IF
			NOT stMqttSettings.bActive
			OR NOT stMqttSettings.bSocketConnection
		THEN
			iState := C_STARTUP;
		END_IF;

	(* read next remaining length *)
	C_RECEIVE_LENGTH:
		fbSocketReceive(
			bExecute := FALSE
		);

		fbSocketReceive(
			sSrvNetId	:= '',
			hSocket		:= stMqttSettings.hSocket,
			cbLen		:= 1,
			pDest		:= ADR(stReceiveBuffer.arMqttData),
			bExecute 	:= TRUE
		);

		iState := C_RECEIVE_LENGTH_WAIT;

	(* wait for remaining length *)
	C_RECEIVE_LENGTH_WAIT:
		fbSocketReceive(
			bExecute := FALSE
		);

		IF
			NOT fbSocketReceive.bBusy
			AND NOT fbSocketReceive.bError
			AND fbSocketReceive.nRecBytes = 1
		THEN
			stMqttSettings.stMqttReceivedTelegram.arMqttData[1 + iLengthPosition] := stReceiveBuffer.arMqttData[0];

			IF stMqttSettings.stMqttReceivedTelegram.arMqttData[1 + iLengthPosition].7 = 1 THEN
				(* read next length byte *)
				iLengthPosition := iLengthPosition + 1;
				iState			:= C_RECEIVE_LENGTH;

				(* Not more the 4 length bytes *)
				IF iLengthPosition > 4 THEN
					iState 					:= C_STARTUP;
					stMqttSettings.bError	:= TRUE;
				END_IF;
			ELSE
				iState := C_RECEIVE_DATA;
			END_IF;
		END_IF;

		IF fbSocketReceive.bError THEN
			iState 					:= C_STARTUP;
			stMqttSettings.bError	:= TRUE;
		END_IF;

		IF
			NOT stMqttSettings.bActive
			OR NOT stMqttSettings.bSocketConnection
		THEN
			iState := C_STARTUP;
		END_IF;

	(* receive remaining data *)
	C_RECEIVE_DATA:
		fbMqttDecodeLength(
			stMqttTelegram	:= stMqttSettings.stMqttReceivedTelegram,
			dwLength		=> dwDataLength
		);

		fbSocketReceive(
			bExecute := FALSE
		);

		fbSocketReceive(
			sSrvNetId	:= '',
			hSocket		:= stMqttSettings.hSocket,
			cbLen		:= dwDataLength,
			pDest		:= ADR(stReceiveBuffer.arMqttData),
			bExecute 	:= TRUE
		);

		iState := C_RECEIVE_DATA_WAIT;

	(* receive *)
	C_RECEIVE_DATA_WAIT:
		fbSocketReceive(
			bExecute := FALSE
		);

		IF
			NOT fbSocketReceive.bBusy
			AND NOT fbSocketReceive.bError
			AND fbSocketReceive.nRecBytes > 0
		THEN
			MEMCPY(
				destAddr	:= ADR(stMqttSettings.stMqttReceivedTelegram.arMqttData[2 + iLengthPosition]),
			    srcAddr		:= ADR(stReceiveBuffer.arMqttData),
				n  			:= fbSocketReceive.nRecBytes
			);
			stMqttSettings.stMqttReceivedTelegram.nDataLength := 2 + iLengthPosition + fbSocketReceive.nRecBytes;

			(* copy last telegram *)
			FC_Mqtt_CopyTelegram_V10(
				stMqttSrcTelegram	:= stMqttSettings.stMqttReceivedTelegram,
				stMqttDestTelegram	:= stMqttSettings.stMqttLastReceivedTelegram,
				stMqttSettings		:= stMqttSettings
			);

			(* check for publish *)
			IF (stMqttSettings.stMqttReceivedTelegram.arMqttData[0] AND 48) = 48 THEN
				ClearReceivedPublishTelegram();

				(* Length MSB/LSB Topic *)
				wTopicLength :=
						SHL(BYTE_TO_WORD(stMqttSettings.stMqttReceivedTelegram.arMqttData[2 + iLengthPosition + 1]), 8) +
						BYTE_TO_WORD(stMqttSettings.stMqttReceivedTelegram.arMqttData[1 + iLengthPosition + 1]);
				wTopicLength := BE16_TO_HOST(wTopicLength);

				(* Copy topic *)
				MEMCPY(
					destAddr	:= ADR(stMqttSettings.stMqttReceivedPublishTelegram.sTopic),
				    srcAddr		:= ADR(stMqttSettings.stMqttReceivedTelegram.arMqttData[3 + iLengthPosition + 1]),
					n  			:= wTopicLength
				);

				(* Copy value *)
				(* value length = remaining data length - length topic value - 2 byte topic length *)
				dwValueLength := dwDataLength - wTopicLength - 2;

				MEMCPY(
					destAddr	:= ADR(stMqttSettings.stMqttReceivedPublishTelegram.sValue),
				    srcAddr		:= ADR(stMqttSettings.stMqttReceivedTelegram.arMqttData[3 + iLengthPosition + 1 + wTopicLength]),
					n  			:= dwValueLength
				);

				stMqttSettings.stMqttReceivedPublishTelegram.bHasData := TRUE;
			END_IF;

			iState	:= C_IDLE;
			bBusy	:= FALSE;
		END_IF;

		IF fbSocketReceive.bError THEN
			iState 					:= C_STARTUP;
			stMqttSettings.bError	:= TRUE;
		END_IF;

		IF
			NOT stMqttSettings.bActive
			OR NOT stMqttSettings.bSocketConnection
		THEN
			iState := C_STARTUP;
		END_IF;

	(* idle *)
	C_IDLE:
		IF
			NOT stMqttSettings.bDisconnect
			AND NOT stMqttSettings.bError
			AND stMqttSettings.bSocketConnection
			AND NOT bBusy
		THEN
			iState := C_RECEIVE_HEADER;
		END_IF;

		IF
			stMqttSettings.bDisconnect
			OR stMqttSettings.bError
			OR NOT stMqttSettings.bSocketConnection
		THEN
			iState := C_STARTUP;
		END_IF;

		(* ensure at least 1 cycle pause *)
		(* bBusy := FALSE; *)

	ELSE
		iState := C_STARTUP;
END_CASE;

(*	END_FUNCTION_BLOCK	*)
END_FUNCTION_BLOCK
ACTION ClearReceivedPublishTelegram:
MEMSET(
	destAddr	:= ADR(stMqttSettings.stMqttReceivedPublishTelegram.sTopic),
	fillByte  	:= 0,
	n			:= 255
);
stMqttSettings.stMqttReceivedPublishTelegram.sTopic := '';

MEMSET(
	destAddr	:= ADR(stMqttSettings.stMqttReceivedPublishTelegram.sValue),
	fillByte  	:= 0,
	n			:= 255
);
stMqttSettings.stMqttReceivedPublishTelegram.sValue := '';

stMqttSettings.stMqttReceivedPublishTelegram.bHasData := FALSE;
END_ACTION

(* POU Intern/FB_Mqtt_DecodeLength_V10, ST *)
(* @NESTEDCOMMENTS := 'Yes' *)
(* @PATH := '\/_Generic\/Mqtt\/Intern' *)
(* @OBJECTFLAGS := '0, 8' *)
(* @SYMFILEFLAGS := '2048' *)
FUNCTION_BLOCK FB_Mqtt_DecodeLength_V10
VAR_INPUT
	stMqttTelegram : ST_MqttTelegram;
END_VAR
VAR_OUTPUT
	dwLength	: DWORD;
	bAmount		: BYTE;
END_VAR
VAR
	index			: INT;
	diMultiplier	: DINT;
	dwValue			: DWORD;
END_VAR
(* @END_DECLARATION := '0' *)
index			:= 0;
diMultiplier	:= 1;
dwValue			:= 0;

REPEAT
	index := index + 1;

	dwValue := dwValue + (stMqttTelegram.arMqttData[index] AND 127) * diMultiplier;
	diMultiplier := diMultiplier * 128;

	IF diMultiplier > 128*128*128 THEN
		dwLength	:= 0;
		bAmount		:= 0;
		RETURN;
	END_IF;
UNTIL stMqttTelegram.arMqttData[index].7 = 0
END_REPEAT;

dwLength	:= dwValue;
bAmount		:= INT_TO_BYTE(index);

(*
multiplier = 1
value = 0

do
	encodedByte = 'next byte from stream'
	value += (encodedByte AND 127) * multiplier
	multiplier *= 128

	if (multiplier > 128*128*128)
		throw Error(Malformed Remaining Length)
while ((encodedByte AND 128) != 0)

*)

(*	END_FUNCTION_BLOCK	*)
END_FUNCTION_BLOCK

(* POU FB_Mqtt_Publish_V10, ST *)
(* @NESTEDCOMMENTS := 'Yes' *)
(* @PATH := '\/_Generic\/Mqtt' *)
(* @OBJECTFLAGS := '0, 8' *)
(* @SYMFILEFLAGS := '2048' *)
FUNCTION_BLOCK FB_Mqtt_Publish_V10
VAR_INPUT
	sTopic	: STRING[255];
	sValue	: STRING[255];
	bRetain	: BOOL := TRUE;
END_VAR
VAR_OUTPUT
	bBusy	: BOOL := FALSE;
END_VAR
VAR_IN_OUT
	stMqttSettings	: ST_MqttSettings;
END_VAR
VAR
	bFirstPublishDone	: BOOL := FALSE;
	bMustPublish		: BOOL := FALSE;
	sLastValue			: STRING[255];
	iState 				: INT := 0;
	iLengthTopic		: INT := 0;
	iLengthValue		: INT := 0;
	wTopicLength		: WORD;
	stMqttTelegram		: ST_MqttTelegram;
	fbMqttEncodeLength	: FB_Mqtt_EncodeLength_V10;
	bLength1			: BYTE;
	bLength2			: BYTE;
	bLength3			: BYTE;
	bLength4			: BYTE;
	bLengthAmount		: BYTE;
END_VAR
VAR CONSTANT
	C_STARTUP			: INT := 0;
	C_BUILD_TELEGRAM	: INT := 100;
	C_SEND_WAIT			: INT := 110;
	C_IDLE				: INT := 500;
END_VAR
(* @END_DECLARATION := '0' *)
CASE iState OF
	C_STARTUP:
		bFirstPublishDone	:= FALSE;
		bBusy				:= FALSE;

		IF stMqttSettings.bValidConnection THEN
			iState := C_IDLE;
		END_IF;

	(* build publish telegram *)
	C_BUILD_TELEGRAM:
		bBusy := TRUE;
		iLengthTopic := LEN(sTopic);
		iLengthValue := LEN(sValue);

		FC_Mqtt_ClearTelegram_V10(
			stMqttTelegram	:= stMqttTelegram,
			stMqttSettings	:= stMqttSettings
		);

		wTopicLength := iLengthTopic;
		wTopicLength := HOST_TO_BE16(wTopicLength);

		(* Calculate length *)
		(* 2 byte length topic, x byte length topic, x byte length value *)
		fbMqttEncodeLength(
			dwLength := 2 + iLengthTopic + iLengthValue,
			bLength1 => bLength1,
			bLength2 => bLength2,
			bLength3 => bLength3,
			bLength4 => bLength4,
			bAmount	 => bLengthAmount
		);

		(* MQTT Control Packet type, no DUP, no QoS, Retain *)
		stMqttTelegram.arMqttData[0] := 48;
		IF bRetain THEN
			stMqttTelegram.arMqttData[0].0 := 1;
		END_IF;

		(* Remaining Length *)
		CASE bLengthAmount OF
			1:
				stMqttTelegram.arMqttData[1] := bLength1;

			2:
				stMqttTelegram.arMqttData[1] := bLength1;
				stMqttTelegram.arMqttData[2] := bLength2;

			3:
				stMqttTelegram.arMqttData[1] := bLength1;
				stMqttTelegram.arMqttData[2] := bLength2;
				stMqttTelegram.arMqttData[3] := bLength3;

			4:
				stMqttTelegram.arMqttData[1] := bLength1;
				stMqttTelegram.arMqttData[2] := bLength2;
				stMqttTelegram.arMqttData[3] := bLength3;
				stMqttTelegram.arMqttData[4] := bLength4;

			ELSE
				iState 					:= C_STARTUP;
				stMqttSettings.bError	:= TRUE;
		END_CASE;

		(* Length MSB Topic *)
		stMqttTelegram.arMqttData[1 + bLengthAmount] := WORD_TO_BYTE(wTopicLength);
		(* Length LSB Topic *)
		stMqttTelegram.arMqttData[2 + bLengthAmount] := WORD_TO_BYTE(SHR(wTopicLength, 8));

		(* Add topic *)
		MEMCPY(
			destAddr	:= ADR(stMqttTelegram.arMqttData[3 + bLengthAmount]),
		    srcAddr		:= ADR(sTopic),
			n  			:= iLengthTopic
		);

		(* Add Payload *)
		MEMCPY(
			destAddr	:= ADR(stMqttTelegram.arMqttData[3 + bLengthAmount + iLengthTopic]),
		    srcAddr		:= ADR(sValue),
			n  			:= iLengthValue
		);

		(* 1 byte header, x byte variable length, 2 byte topic lenght, x byte topic, x byte value *)
		stMqttTelegram.nDataLength := 1 + bLengthAmount + 2 + iLengthTopic + iLengthValue;

		iState := C_SEND_WAIT;

	(* send telegram *)
	C_SEND_WAIT:
		IF stMqttSettings.stMqttSendTelegram.nDataLength = 0 THEN
			FC_Mqtt_CopyTelegram_V10(
				stMqttSrcTelegram	:= stMqttTelegram,
				stMqttDestTelegram	:= stMqttSettings.stMqttSendTelegram,
				stMqttSettings		:= stMqttSettings
			);

			iState				:= C_IDLE;
			bFirstPublishDone	:= TRUE;
			sLastValue			:= sValue;
		END_IF;

		IF NOT stMqttSettings.bValidConnection THEN
			iState := C_STARTUP;
		END_IF;

	(* idle *)
	C_IDLE:
		bBusy 			:= FALSE;
		bMustPublish 	:= sLastValue <> sValue;

		IF
			stMqttSettings.bValidConnection
			AND (
				bMustPublish
				OR NOT bFirstPublishDone
			)
		THEN
			iState := C_BUILD_TELEGRAM;
		END_IF;

		IF NOT stMqttSettings.bValidConnection THEN
			iState := C_STARTUP;
		END_IF;

	ELSE
		iState := C_STARTUP;
END_CASE;

(*	END_FUNCTION_BLOCK	*)
END_FUNCTION_BLOCK

(* POU Thermocontrol, ST *)
PROGRAM Thermocontrol
VAR
	period_sec		: INT:=120;  (* Частота работы термостата, секунды*)
	gisterezis		: REAL:=0.2; (*Гистерезис термостата, градусы цельсия *)
	Timer1			: TON;
	Timer1Q			: BOOL;
	state			: INT:=0;
	 tTimerValue		: TIME;
END_VAR
tTimerValue := DINT_TO_TIME(period_sec*1000);

CASE state OF
0:
	IF (iobroker.First_floor_temp > iobroker.First_floor_temp_target+gisterezis ) THEN
		HW_heat_first_floor:=FALSE;
	END_IF

	IF (iobroker.First_floor_temp <  iobroker.First_floor_temp_target-gisterezis ) THEN
		HW_heat_first_floor:=TRUE;
	END_IF

	state:=1;

1:
	IF (iobroker.Second_floor_temp > iobroker.Second_floor_temp_target+gisterezis ) THEN
		HW_heat_Second_floor:=FALSE;
	END_IF

	IF (iobroker.Second_floor_temp <  iobroker.Second_floor_temp_target-gisterezis ) THEN
		HW_heat_Second_floor:=TRUE;
	END_IF

	state:=2;
2:
	IF (iobroker.Sport_temp > iobroker.Sport_temp_target+gisterezis ) THEN
		HW_heat_sport:=FALSE;
	END_IF

	IF (iobroker.Sport_temp <  iobroker.Sport_temp_target-gisterezis ) THEN
		HW_heat_sport:=TRUE;
	END_IF

	state:=3;

3:
	IF (iobroker.Sauna_temp > iobroker.Sauna_temp_target+gisterezis ) THEN
		HW_heat_Sauna:=FALSE;
	END_IF

	IF (iobroker.Sauna_temp <  iobroker.Sauna_temp_target-gisterezis ) THEN
		HW_heat_Sauna:=TRUE;
	END_IF

	state:=4;

4:
	IF (iobroker.Underfloor_temp > iobroker.Underfloor_temp_target+gisterezis AND iobroker.Underfloor_humidity < iobroker.Underfloor_humidity_target-1 ) THEN
		HW_heat_underfloor:=FALSE;
	END_IF

	IF (iobroker.Underfloor_temp <  iobroker.Underfloor_temp_target-gisterezis OR iobroker.Underfloor_humidity > iobroker.Underfloor_humidity_target+1) THEN
		HW_heat_Underfloor:=TRUE;
	END_IF

	state:=100;



100:


	Timer1(IN:=NOT Timer1Q , PT:=tTimerValue , Q=>Timer1Q , ET=> );
		IF timer1.q THEN

		state:=0;
		END_IF



END_CASE
END_PROGRAM

(* POU VentControl, ST *)
PROGRAM VentControl
VAR
	Temperature_max_to_heat	: REAL:=17;		(* Максимальная температура наружнего воздуха при которой разрешено включать воздухонагреватель*)
	gisterezis				: REAL:=0.2;	(* Гистерезис  разрешения включения воздухонагревателя, градусы цельсия *)
	vent_valve_opened	 	: BOOL:=FALSE;	(*После перезагрузки ПЛК считаем что приточный клапан закрыт *)
	Period_start_delay		: INT:=60; 	(* Время задержки включения вентилятора после сигнала на открытие приточного клапана, сек *)
	Period_stop_delay		: INT:=60;		(* Время задержки отключения вентилятора после сигнала на останов вентиляции - для остужения разогретых ТЭНов воздухонагревателя, сек *)
	Timer1					: TON;		(* Таймер задержки включения вентилятора после сигнала на открытие приточного клапана *)
	Timer2					: TON;		(* Таймер задержки отключения вентилятора после сигнала на останов вентиляции - для остужения разогретых ТЭНов воздухонагревателя *)
	Timer1Q					: BOOL;
	Timer2Q					: BOOL;
	tTimerValue1				: TIME;
	tTimerValue2				: TIME;
END_VAR
tTimerValue1 := DINT_TO_TIME(Period_start_delay*1000);
tTimerValue2 := DINT_TO_TIME(Period_stop_delay*1000);

IF (iobroker.Vent=FALSE) THEN
	HW_vent_in_heat := FALSE;
	vent_valve_opened := FALSE;
	HW_vent_valve_input:=FALSE;
	Timer2(IN:=NOT Timer2Q , PT:=tTimerValue2 , Q=>Timer2Q , ET=> );
	IF timer2q THEN
		HW_trans_power:=FALSE;
	END_IF


ELSE
	HW_vent_valve_input:=TRUE;
	HW_vent_valve_output:=TRUE;

	IF (vent_valve_opened = FALSE) THEN
		Timer1(IN:=NOT Timer1Q , PT:=tTimerValue1 , Q=>Timer1Q , ET=> );
		IF timer1.q THEN
			vent_valve_opened := TRUE;
		END_IF
	END_IF

	IF (vent_valve_opened=TRUE) THEN
		HW_trans_power:=TRUE;
(*		IF (HW_vent_reay_pressure=TRUE) THEN	*)

			IF (iobroker.Vent_heat=2) THEN
				IF (iobroker.Street_temp < Temperature_max_to_heat-gisterezis) THEN
					HW_vent_in_heat:=TRUE;
					IF (iobroker.Vent_heat_level=TRUE) THEN
						HW_vent_in_heat_level:=TRUE;
					END_IF
				END_IF
				IF (iobroker.Street_temp > Temperature_max_to_heat+gisterezis) THEN
					HW_vent_in_heat:=FALSE;
				END_IF
			ELSE
				IF (iobroker.Vent_heat=1) THEN
					HW_vent_in_heat:=TRUE;
					IF (iobroker.Vent_heat_level=TRUE) THEN
						HW_vent_in_heat_level:=TRUE;
					ELSE
						HW_vent_in_heat_level:=FALSE;
					END_IF
				END_IF
				IF (iobroker.Vent_heat=0) THEN
					HW_vent_in_heat:=FALSE;
				END_IF
			END_IF
(*		END_IF   *)(*vent_relay_pressure*)
	END_IF (*vent_valve_opened*)
END_IF (*Vent*)
END_PROGRAM

(* POU VentPower, ST *)
PROGRAM VentPower
VAR
	Vent_power			: REAL:=30;  (* После перезагрузки ПЛК задаём начальную мощность условных 30%  *)
	CO2_old				: REAL:=410; (* После перезагрузки ПЛК задаём принудительно последнее значение CO2 = 410 (абсолютно свежий воздух) *)
	Period_vent_switch	: INT:=60; (* Частота переключения режимов работы вентилятора по показаниям датчиков CO2, секунды*)
	Timer1				: TON;
	Timer1Q				: BOOL;
	count				: INT:=0;
	CO2_max			: REAL;
	tTimerValue			: TIME;

END_VAR
tTimerValue := DINT_TO_TIME(Period_vent_switch*1000);

IF (iobroker.Vent =TRUE  ) THEN

	Timer1(IN:=NOT Timer1Q , PT:=tTimerValue , Q=>Timer1Q , ET=> );

	IF timer1.q THEN
	CO2_max:=MAX (iobroker.First_floor_CO2, iobroker.Second_floor_CO2);

	IF (  (CO2_max >=  CO2_old-10 )  AND ( CO2_max >  INT_TO_REAL(iobroker.Target_CO2)*1.05 ) ) THEN
			Vent_power:=Vent_power+5;
		END_IF
		count:=count+1;

		IF (count = 2)	THEN
			IF (  CO2_max <=  INT_TO_REAL(iobroker.Target_CO2)*0.99) THEN
				Vent_power:=Vent_power-1;
			END_IF
		count:=1;
		END_IF

		IF (Vent_power>80) THEN
			Vent_power:=80;
		END_IF
		IF(Vent_power<20) THEN
			Vent_power:=20;
		END_IF

		IF (Vent_Power > 75  ) THEN

			iobroker.Vent_input_level:=200;	(*200 м. куб в час при подаче напряжения на вентилятор  220V *)
			HW_vent_in_trans_160_220:=FALSE;
			HW_vent_in_trans_LO_HI:=FALSE;


			ELSIF (Vent_Power>50 ) THEN

				iobroker.Vent_input_level:=180; (*200 м. куб в час при подаче напряжения на вентилятор 220V *)
				HW_vent_in_trans_160_220:=FALSE;
				HW_vent_in_trans_LO_HI:=FALSE;

			ELSIF (Vent_Power>35 AND Vent_Power<=50) THEN

					iobroker.Vent_input_level:=150; (* 150 м. куб в час при подаче напряжения на вентилятор160V *)
					HW_vent_in_trans_160_220:=TRUE;
					HW_vent_in_trans_LO_HI:=FALSE;

			ELSIF (Vent_Power>25 AND Vent_Power<=35) THEN

					iobroker.Vent_input_level:=110; (* 110 м. куб в час при подаче напряжения на вентилятор 130V *)
					HW_vent_in_trans_105_130:=FALSE;
					HW_vent_in_trans_LO_HI:=TRUE;


			ELSE
				iobroker.Vent_input_level:=80; (* 80 м. куб в час при подаче напряжения на вентилятор 105V *)
				HW_vent_in_trans_105_130:=TRUE;
				HW_vent_in_trans_LO_HI:=TRUE;


			END_IF

			CO2_old:=CO2_max;

		END_IF	(* Timer1 *)

	ELSE	 (* Vent=TRUE*)


		iobroker.Vent_input_level:=0;

END_IF   (* Vent=TRUE*)
END_PROGRAM

(* POU Poliv, ST *)
PROGRAM Poliv
VAR
	Period_pomp_garden_delay	: INT:=15;				(* Задержка включения насоса после сигнала на открытие клапана=15 сек. *)

 	 tTimerValue_zapad			: TIME;
	Timer_poliv_zapad			: TON;
	Timer_poliv_zapadQ			:  BOOL;

	tTimerValue_terrasa			: TIME;
	Timer_poliv_terrasa			: TON;
	Timer_poliv_terrasaQ			:  BOOL;

	 tTimerValue_south			: TIME;
	Timer_poliv_south				: TON;
	Timer_poliv_southQ			:  BOOL;

	TON_pomp_garden			: TON ;
	pomp_garden_start			: BOOL;

	tTimerValue					: TIME;
END_VAR
tTimerValue := DINT_TO_TIME(Period_pomp_garden_delay*1000);


Timer_poliv_zapad();
Timer_poliv_terrasa();
Timer_poliv_south();

IF (iobroker.Poliv_zapad = TRUE ) THEN
	tTimerValue_zapad := DINT_TO_TIME(iobroker.Poliv_zapad_minutes*60*1000);
	HW_poliv_zapad	:=	TRUE;
	Timer_poliv_zapad(IN:=NOT Timer_poliv_zapadQ , PT:=tTimerValue_zapad , Q=>Timer_poliv_zapadQ , ET=> );
END_IF
IF (iobroker.Poliv_zapad = FALSE ) THEN
	HW_poliv_zapad	:=	FALSE;
	Timer_poliv_zapadQ := FALSE;
	Timer_poliv_zapad(IN:=FALSE , PT:=T#0ms , Q=>Timer_poliv_zapadQ , ET=> );
END_IF
IF Timer_poliv_zapad.q THEN
	iobroker.Poliv_zapad := FALSE;
	HW_poliv_zapad	:=	FALSE;
END_IF


IF (iobroker.Poliv_terrasa = TRUE ) THEN
	tTimerValue_terrasa := DINT_TO_TIME(iobroker.Poliv_terrasa_minutes*60*1000);
	HW_poliv_terrasa	:=	TRUE;
	Timer_poliv_terrasa(IN:=NOT Timer_poliv_terrasaQ , PT:=tTimerValue_terrasa , Q=>Timer_poliv_terrasaQ , ET=> );
END_IF
IF (iobroker.Poliv_terrasa = FALSE ) THEN
	HW_poliv_terrasa	:=	FALSE;
	Timer_poliv_terrasaQ := FALSE;
	Timer_poliv_terrasa(IN:=FALSE , PT:=T#0ms , Q=>Timer_poliv_terrasaQ , ET=> );
END_IF
IF Timer_poliv_terrasa.q THEN
	iobroker.Poliv_terrasa := FALSE;
	HW_poliv_zapad	:=	FALSE;
END_IF

IF (iobroker.Poliv_south = TRUE ) THEN
	tTimerValue_south := DINT_TO_TIME(iobroker.Poliv_south_minutes*60*1000);
	HW_poliv_south	:=	TRUE;
	Timer_poliv_south(IN:=NOT Timer_poliv_southQ , PT:=tTimerValue_south , Q=>Timer_poliv_southQ , ET=> );
END_IF
IF (iobroker.Poliv_south = FALSE ) THEN
	HW_poliv_south	:=	FALSE;
	Timer_poliv_southQ := FALSE;
	Timer_poliv_south(IN:=FALSE , PT:=T#0ms , Q=>Timer_poliv_southQ , ET=> );
END_IF
IF Timer_poliv_south.q THEN
	iobroker.Poliv_south := FALSE;
	HW_poliv_south	:=	FALSE;
END_IF

IF ((HW_poliv_zapad=TRUE OR HW_poliv_terrasa=TRUE 	OR HW_poliv_south =	TRUE) AND (HW_pomp_Garden=FALSE)  )  THEN
	pomp_garden_start			:=TRUE;
END_IF


TON_pomp_garden(IN := pomp_garden_start, PT:= tTimerValue);
iobroker.Pomp_garden	 	:= TON_pomp_garden.Q;
HW_Pomp_garden		:= TON_pomp_garden.Q;

IF ((HW_poliv_zapad=FALSE AND HW_poliv_terrasa=FALSE 	AND HW_poliv_south = FALSE))   THEN
	pomp_garden_start		:= FALSE;
	iobroker.Pomp_garden	 	:= FALSE;
	HW_Pomp_garden		:= FALSE;
END_IF
END_PROGRAM

(* POU FB_Mqtt_Subscribe_V10, ST *)
(* @NESTEDCOMMENTS := 'Yes' *)
(* @PATH := '\/_Generic\/Mqtt' *)
(* @OBJECTFLAGS := '0, 8' *)
(* @SYMFILEFLAGS := '2048' *)
FUNCTION_BLOCK FB_Mqtt_Subscribe_V10
VAR_INPUT
	sTopic	: STRING[255];
	bAccept	: BOOL := FALSE; (* When false, subscribe but do not set bNewValue output *)
END_VAR
VAR_OUTPUT
	sValue		: STRING[255];
	bNewValue	: BOOL := FALSE;
	bBusy		: BOOL := FALSE;
END_VAR
VAR_IN_OUT
	stMqttSettings	: ST_MqttSettings;
END_VAR
VAR
	iState 				: INT := 0;
	bSubscribeSent		: BOOL := FALSE;
	bSubAckReceived		: BOOL := FALSE;
	iTopicLength		: INT := 0;
	wTopicLength		: WORD;
	stMqttTelegram		: ST_MqttTelegram;
	fbMqttEncodeLength	: FB_Mqtt_EncodeLength_V10;
	bLength1			: BYTE;
	bLength2			: BYTE;
	bLength3			: BYTE;
	bLength4			: BYTE;
	bLengthAmount		: BYTE;

	wPackageIdentifier			: WORD;
	wTelegramPackageIdentifier	: WORD;
END_VAR
VAR CONSTANT
	C_STARTUP			: INT := 0;
	C_BUILD_TELEGRAM	: INT := 100;
	C_SEND_WAIT			: INT := 110;
	C_CHECK_TELEGRAM	: INT := 200;
	C_IDLE				: INT := 500;
END_VAR

(* @END_DECLARATION := '0' *)
CASE iState OF
	C_STARTUP:
		wPackageIdentifier 	:= 0;
		bSubscribeSent		:= FALSE;
		bSubAckReceived		:= FALSE;
		bNewValue			:= FALSE;
		sValue 				:= '';
		bBusy				:= FALSE;

		IF stMqttSettings.bValidConnection THEN
			iState := C_IDLE;
		END_IF;

	(* build publish telegram *)
	C_BUILD_TELEGRAM:
		bBusy 								:= TRUE;
		wPackageIdentifier 					:= stMqttSettings.wPackageIdentifier;
		stMqttSettings.wPackageIdentifier 	:= stMqttSettings.wPackageIdentifier + 1;
		iTopicLength						:= LEN(sTopic);

		FC_Mqtt_ClearTelegram_V10(
			stMqttTelegram	:= stMqttTelegram,
			stMqttSettings	:= stMqttSettings
		);

		wTopicLength := iTopicLength;
		wTopicLength := HOST_TO_BE16(wTopicLength);

		wTelegramPackageIdentifier := HOST_TO_BE16(wPackageIdentifier);

		(* Calculate length *)
		(* 2 byte package identifier, 2 byte length topic, x byte length topic, 1 byte QoS *)
		fbMqttEncodeLength(
			dwLength := 2 + 2 + iTopicLength + 1,
			bLength1 => bLength1,
			bLength2 => bLength2,
			bLength3 => bLength3,
			bLength4 => bLength4,
			bAmount	 => bLengthAmount
		);

		(* MQTT Control Packet type *)
		stMqttTelegram.arMqttData[0] := 130;

		(* Remaining Length *)
		CASE bLengthAmount OF
			1:
				stMqttTelegram.arMqttData[1] := bLength1;

			2:
				stMqttTelegram.arMqttData[1] := bLength1;
				stMqttTelegram.arMqttData[2] := bLength2;

			3:
				stMqttTelegram.arMqttData[1] := bLength1;
				stMqttTelegram.arMqttData[2] := bLength2;
				stMqttTelegram.arMqttData[3] := bLength3;

			4:
				stMqttTelegram.arMqttData[1] := bLength1;
				stMqttTelegram.arMqttData[2] := bLength2;
				stMqttTelegram.arMqttData[3] := bLength3;
				stMqttTelegram.arMqttData[4] := bLength4;

			ELSE
				iState 					:= C_STARTUP;
				stMqttSettings.bError	:= TRUE;
		END_CASE;

		(* Packet Identifier MSB *)
		stMqttTelegram.arMqttData[1 + bLengthAmount] := WORD_TO_BYTE(wTelegramPackageIdentifier);
		(* Packet Identifier LSB *)
		stMqttTelegram.arMqttData[2 + bLengthAmount] := WORD_TO_BYTE(SHR(wTelegramPackageIdentifier, 8));
		(* Length MSB Topic *)
		stMqttTelegram.arMqttData[3 + bLengthAmount] := WORD_TO_BYTE(wTopicLength);
		(* Length MSB Topic *)
		stMqttTelegram.arMqttData[4 + bLengthAmount] := WORD_TO_BYTE(SHR(wTopicLength, 8));

		(* Add topic *)
		MEMCPY(
			destAddr	:= ADR(stMqttTelegram.arMqttData[5 + bLengthAmount]),
		    srcAddr		:= ADR(sTopic),
			n  			:= iTopicLength
		);

		(* 1 byte header, x byte variable length, 2 byte package identifier, 2 byte topic lenght, x byte topic, 1 byte QoS *)
		stMqttTelegram.nDataLength := 1 + bLengthAmount + 2 + 2 + iTopicLength + 1;

		iState := C_SEND_WAIT;

	(* send telegram *)
	C_SEND_WAIT:
		IF stMqttSettings.stMqttSendTelegram.nDataLength = 0 THEN
			FC_Mqtt_CopyTelegram_V10(
				stMqttSrcTelegram	:= stMqttTelegram,
				stMqttDestTelegram	:= stMqttSettings.stMqttSendTelegram,
				stMqttSettings		:= stMqttSettings
			);

			bSubscribeSent	:= TRUE;
			iState			:= C_IDLE;
		END_IF;

		IF NOT stMqttSettings.bValidConnection THEN
			iState := C_STARTUP;
		END_IF;

	(* check telegram *)
	C_CHECK_TELEGRAM:
		bBusy 			:= TRUE;

		IF
			stMqttSettings.stMqttReceivedPublishTelegram.bHasData
			AND stMqttSettings.stMqttReceivedPublishTelegram.sTopic = sTopic
		THEN
			FC_Mqtt_ClearTelegram_V10(
				stMqttTelegram	:= stMqttSettings.stMqttReceivedTelegram,
				stMqttSettings	:= stMqttSettings
			);
			stMqttSettings.stMqttReceivedPublishTelegram.bHasData := FALSE;

			sValue		:= stMqttSettings.stMqttReceivedPublishTelegram.sValue;
			bNewValue 	:= TRUE;
		END_IF;

		iState := C_IDLE;

	(* idle *)
	C_IDLE:
		bBusy 		:= FALSE;
		bNewValue	:= FALSE;

		IF
			stMqttSettings.bValidConnection
			AND NOT bSubscribeSent
			AND NOT bSubAckReceived
		THEN
			iState := C_BUILD_TELEGRAM;
		END_IF;

		(* Check for correct SubAck *)
		IF
			bSubscribeSent
			AND stMqttSettings.stMqttReceivedTelegram.nDataLength = 5
			AND stMqttSettings.stMqttReceivedTelegram.arMqttData[0] = 144
			AND stMqttSettings.stMqttReceivedTelegram.arMqttData[1] = 3
			AND stMqttSettings.stMqttReceivedTelegram.arMqttData[2] = WORD_TO_BYTE(wTelegramPackageIdentifier)
			AND stMqttSettings.stMqttReceivedTelegram.arMqttData[3] = WORD_TO_BYTE(SHR(wTelegramPackageIdentifier, 8))
			AND stMqttSettings.stMqttReceivedTelegram.arMqttData[4] = 0
		THEN
			FC_Mqtt_ClearTelegram_V10(
				stMqttTelegram	:= stMqttSettings.stMqttReceivedTelegram,
				stMqttSettings	:= stMqttSettings
			);
			bSubAckReceived := TRUE;
		END_IF;

		(* Check for error SubAck *)
		IF
			bSubscribeSent
			AND stMqttSettings.stMqttReceivedTelegram.nDataLength = 5
			AND stMqttSettings.stMqttReceivedTelegram.arMqttData[0] = 144
			AND stMqttSettings.stMqttReceivedTelegram.arMqttData[1] = 3
			AND stMqttSettings.stMqttReceivedTelegram.arMqttData[2] = WORD_TO_BYTE(wTelegramPackageIdentifier)
			AND stMqttSettings.stMqttReceivedTelegram.arMqttData[3] = WORD_TO_BYTE(SHR(wTelegramPackageIdentifier, 8))
			AND stMqttSettings.stMqttReceivedTelegram.arMqttData[4].7 = 1
		THEN
			stMqttSettings.bError := TRUE;
		END_IF;

		(* Check for publish *)
		IF
			bSubAckReceived
			AND stMqttSettings.stMqttReceivedPublishTelegram.bHasData
			AND bAccept
		THEN
			iState := C_CHECK_TELEGRAM;
		END_IF;

		IF NOT stMqttSettings.bValidConnection THEN
			iState := C_STARTUP;
		END_IF;

	ELSE
		iState := C_STARTUP;
END_CASE

(*	END_FUNCTION_BLOCK	*)
END_FUNCTION_BLOCK
